LIN {X -0.090,Y -532.031,Z 1144.398,A 0.000,B 0.000,C 90.000,E1 287.692} C_DIS
LIN {X -0.142,Y -531.447,Z 1144.390,A 0.000,B 0.000,C 90.000,E1 286.260} C_DIS
LIN {X -0.170,Y -530.686,Z 1144.381,A 0.000,B 0.000,C 90.000,E1 284.537} C_DIS
LIN {X 0.098,Y -529.977,Z 1144.374,A 0.000,B 0.000,C 90.000,E1 283.355} C_DIS
LIN {X -0.145,Y -528.701,Z 1144.361,A 0.000,B 0.000,C 90.000,E1 281.074} C_DIS
LIN {X 0.034,Y -527.720,Z 1144.352,A 0.000,B 0.000,C 90.000,E1 279.321} C_DIS
LIN {X 0.037,Y -526.581,Z 1144.341,A 0.000,B 0.000,C 90.000,E1 277.296} C_DIS
LIN {X -0.057,Y -525.479,Z 1144.329,A 0.000,B 0.000,C 90.000,E1 275.277} C_DIS
LIN {X 0.247,Y -524.532,Z 1144.316,A 0.000,B 0.000,C 90.000,E1 272.922} C_DIS
LIN {X 0.030,Y -523.822,Z 1144.307,A 0.000,B 0.000,C 90.000,E1 271.203} C_DIS
LIN {X -0.209,Y -523.045,Z 1144.297,A 0.000,B 0.000,C 90.000,E1 269.484} C_DIS
LIN {X 0.023,Y -522.107,Z 1144.286,A 0.000,B 0.000,C 90.000,E1 267.421} C_DIS
LIN {X -0.216,Y -521.259,Z 1144.276,A 0.000,B 0.000,C 90.000,E1 265.698} C_DIS
LIN {X 0.175,Y -520.707,Z 1144.271,A 0.000,B 0.000,C 90.000,E1 264.780} C_DIS
LIN {X 0.024,Y -519.813,Z 1144.265,A 0.000,B 0.000,C 90.000,E1 263.628} C_DIS
LIN {X -0.168,Y -518.040,Z 1144.255,A 0.000,B 0.000,C 90.000,E1 261.894} C_DIS
LIN {X 0.162,Y -515.646,Z 1144.242,A 0.000,B 0.000,C 90.000,E1 259.511} C_DIS
LIN {X 0.113,Y -514.734,Z 1144.237,A 0.000,B 0.000,C 90.000,E1 258.634} C_DIS
LIN {X 0.008,Y -513.326,Z 1144.229,A 0.000,B 0.000,C 90.000,E1 257.173} C_DIS
LIN {X 0.011,Y -511.181,Z 1144.216,A 0.000,B 0.000,C 90.000,E1 254.810} C_DIS
LIN {X 0.078,Y -509.858,Z 1144.207,A 0.000,B 0.000,C 90.000,E1 253.323} C_DIS
LIN {X 0.266,Y -508.448,Z 1144.199,A 0.000,B 0.000,C 90.000,E1 251.819} C_DIS
LIN {X -0.151,Y -507.301,Z 1144.193,A 0.000,B 0.000,C 90.000,E1 250.678} C_DIS
LIN {X -0.143,Y -505.111,Z 1144.181,A 0.000,B 0.000,C 90.000,E1 248.592} C_DIS
LIN {X 0.211,Y -503.811,Z 1144.174,A 0.000,B 0.000,C 90.000,E1 247.358} C_DIS
LIN {X 0.078,Y -502.418,Z 1144.168,A 0.000,B 0.000,C 90.000,E1 246.177} C_DIS
LIN {X 0.129,Y -500.836,Z 1144.161,A 0.000,B 0.000,C 90.000,E1 244.973} C_DIS
LIN {X -0.230,Y -498.804,Z 1144.153,A 0.000,B 0.000,C 90.000,E1 243.512} C_DIS
LIN {X -0.124,Y -496.185,Z 1144.143,A 0.000,B 0.000,C 90.000,E1 241.691} C_DIS
LIN {X 0.057,Y -494.353,Z 1144.136,A 0.000,B 0.000,C 90.000,E1 240.461} C_DIS
LIN {X 0.033,Y -491.924,Z 1144.128,A 0.000,B 0.000,C 90.000,E1 238.948} C_DIS
LIN {X -0.041,Y -490.014,Z 1144.121,A 0.000,B 0.000,C 90.000,E1 237.740} C_DIS
LIN {X 0.192,Y -487.119,Z 1144.111,A 0.000,B 0.000,C 90.000,E1 235.881} C_DIS
LIN {X -0.043,Y -484.123,Z 1144.100,A 0.000,B 0.000,C 90.000,E1 234.069} C_DIS
LIN {X -0.266,Y -481.618,Z 1144.092,A 0.000,B 0.000,C 90.000,E1 232.557} C_DIS
LIN {X -0.058,Y -478.479,Z 1144.082,A 0.000,B 0.000,C 90.000,E1 230.678} C_DIS
LIN {X -0.148,Y -475.794,Z 1144.073,A 0.000,B 0.000,C 90.000,E1 229.138} C_DIS
LIN {X 0.171,Y -472.605,Z 1144.063,A 0.000,B 0.000,C 90.000,E1 227.229} C_DIS
LIN {X -0.067,Y -466.133,Z 1144.040,A 0.000,B 0.000,C 90.000,E1 223.176} C_DIS
LIN {X 0.091,Y -463.472,Z 1144.028,A 0.000,B 0.000,C 90.000,E1 220.943} C_DIS
LIN {X -0.133,Y -461.119,Z 1144.015,A 0.000,B 0.000,C 90.000,E1 218.749} C_DIS
LIN {X 0.111,Y -458.835,Z 1144.001,A 0.000,B 0.000,C 90.000,E1 216.171} C_DIS
LIN {X -0.031,Y -455.791,Z 1143.971,A 0.000,B 0.000,C 90.000,E1 210.747} C_DIS
LIN {X 0.088,Y -455.692,Z 1143.958,A 0.000,B 0.000,C 90.000,E1 208.487} C_DIS
LIN {X 0.068,Y -456.850,Z 1143.944,A 0.000,B 0.000,C 90.000,E1 205.924} C_DIS
LIN {X -0.111,Y -458.875,Z 1143.933,A 0.000,B 0.000,C 90.000,E1 204.027} C_DIS
LIN {X 0.171,Y -461.835,Z 1143.923,A 0.000,B 0.000,C 90.000,E1 202.078} C_DIS
LIN {X -0.117,Y -467.069,Z 1143.909,A 0.000,B 0.000,C 90.000,E1 199.577} C_DIS
LIN {X 0.019,Y -474.758,Z 1143.893,A 0.000,B 0.000,C 90.000,E1 196.732} C_DIS
LIN {X 0.039,Y -483.007,Z 1143.879,A 0.000,B 0.000,C 90.000,E1 194.245} C_DIS
LIN {X -0.161,Y -490.571,Z 1143.867,A 0.000,B 0.000,C 90.000,E1 192.119} C_DIS
LIN {X -0.200,Y -496.173,Z 1143.859,A 0.000,B 0.000,C 90.000,E1 190.602} C_DIS
LIN {X 0.210,Y -502.992,Z 1143.849,A 0.000,B 0.000,C 90.000,E1 188.746} C_DIS
LIN {X -0.174,Y -508.766,Z 1143.840,A 0.000,B 0.000,C 90.000,E1 187.296} C_DIS
LIN {X -0.020,Y -514.520,Z 1143.832,A 0.000,B 0.000,C 90.000,E1 185.796} C_DIS
LIN {X 0.198,Y -520.225,Z 1143.824,A 0.000,B 0.000,C 90.000,E1 184.302} C_DIS
LIN {X -0.001,Y -525.916,Z 1143.816,A 0.000,B 0.000,C 90.000,E1 182.865} C_DIS
LIN {X -0.163,Y -533.787,Z 1143.805,A 0.000,B 0.000,C 90.000,E1 180.859} C_DIS
LIN {X -0.160,Y -539.409,Z 1143.797,A 0.000,B 0.000,C 90.000,E1 179.427} C_DIS
LIN {X -0.042,Y -545.053,Z 1143.789,A 0.000,B 0.000,C 90.000,E1 177.993} C_DIS
LIN {X 0.235,Y -551.836,Z 1143.780,A 0.000,B 0.000,C 90.000,E1 176.274} C_DIS
LIN {X 0.255,Y -559.740,Z 1143.769,A 0.000,B 0.000,C 90.000,E1 174.318} C_DIS
LIN {X 0.285,Y -565.342,Z 1143.761,A 0.000,B 0.000,C 90.000,E1 172.932} C_DIS
LIN {X -0.147,Y -570.919,Z 1143.753,A 0.000,B 0.000,C 90.000,E1 171.602} C_DIS
LIN {X -0.038,Y -575.313,Z 1143.747,A 0.000,B 0.000,C 90.000,E1 170.500} C_DIS
LIN {X 0.132,Y -579.671,Z 1143.741,A 0.000,B 0.000,C 90.000,E1 169.398} C_DIS
LIN {X 0.137,Y -585.038,Z 1143.734,A 0.000,B 0.000,C 90.000,E1 168.049} C_DIS
LIN {X 0.240,Y -590.168,Z 1143.726,A 0.000,B 0.000,C 90.000,E1 166.700} C_DIS
LIN {X 0.150,Y -594.155,Z 1143.720,A 0.000,B 0.000,C 90.000,E1 165.644} C_DIS
LIN {X 0.260,Y -597.917,Z 1143.714,A 0.000,B 0.000,C 90.000,E1 164.574} C_DIS
LIN {X 0.033,Y -603.261,Z 1143.706,A 0.000,B 0.000,C 90.000,E1 163.015} C_DIS
LIN {X 0.184,Y -607.423,Z 1143.698,A 0.000,B 0.000,C 90.000,E1 161.692} C_DIS
LIN {X -0.115,Y -610.638,Z 1143.693,A 0.000,B 0.000,C 90.000,E1 160.678} C_DIS
LIN {X -0.224,Y -614.444,Z 1143.685,A 0.000,B 0.000,C 90.000,E1 159.390} C_DIS
LIN {X -0.269,Y -617.969,Z 1143.678,A 0.000,B 0.000,C 90.000,E1 158.103} C_DIS
LIN {X -0.027,Y -622.096,Z 1143.670,A 0.000,B 0.000,C 90.000,E1 156.538} C_DIS
LIN {X 0.317,Y -626.734,Z 1143.660,A 0.000,B 0.000,C 90.000,E1 154.717} C_DIS
LIN {X 0.137,Y -629.863,Z 1143.653,A 0.000,B 0.000,C 90.000,E1 153.461} C_DIS
LIN {X -0.282,Y -632.833,Z 1143.646,A 0.000,B 0.000,C 90.000,E1 152.231} C_DIS
LIN {X 0.209,Y -635.650,Z 1143.639,A 0.000,B 0.000,C 90.000,E1 150.923} C_DIS
LIN {X 0.198,Y -638.324,Z 1143.632,A 0.000,B 0.000,C 90.000,E1 149.665} C_DIS
LIN {X 0.227,Y -640.892,Z 1143.625,A 0.000,B 0.000,C 90.000,E1 148.408} C_DIS
LIN {X -0.310,Y -642.835,Z 1143.619,A 0.000,B 0.000,C 90.000,E1 147.454} C_DIS
LIN {X 0.003,Y -645.547,Z 1143.611,A 0.000,B 0.000,C 90.000,E1 145.928} C_DIS
LIN {X -0.053,Y -647.723,Z 1143.604,A 0.000,B 0.000,C 90.000,E1 144.689} C_DIS
LIN {X 0.262,Y -650.648,Z 1143.594,A 0.000,B 0.000,C 90.000,E1 142.924} C_DIS
LIN {X -0.006,Y -654.464,Z 1143.582,A 0.000,B 0.000,C 90.000,E1 140.723} C_DIS
LIN {X -0.168,Y -657.760,Z 1143.572,A 0.000,B 0.000,C 90.000,E1 139.013} C_DIS
LIN {X -0.321,Y -661.207,Z 1143.563,A 0.000,B 0.000,C 90.000,E1 137.310} C_DIS
LIN {X 0.053,Y -665.103,Z 1143.552,A 0.000,B 0.000,C 90.000,E1 135.324} C_DIS
LIN {X 0.059,Y -669.952,Z 1143.540,A 0.000,B 0.000,C 90.000,E1 133.137} C_DIS
LIN {X -0.245,Y -674.550,Z 1143.529,A 0.000,B 0.000,C 90.000,E1 131.229} C_DIS
LIN {X 0.115,Y -679.826,Z 1143.517,A 0.000,B 0.000,C 90.000,E1 129.036} C_DIS
LIN {X -0.068,Y -682.910,Z 1143.510,A 0.000,B 0.000,C 90.000,E1 127.855} C_DIS
LIN {X -0.046,Y -686.505,Z 1143.502,A 0.000,B 0.000,C 90.000,E1 126.423} C_DIS
LIN {X 0.011,Y -689.481,Z 1143.496,A 0.000,B 0.000,C 90.000,E1 125.231} C_DIS
LIN {X 0.332,Y -692.949,Z 1143.488,A 0.000,B 0.000,C 90.000,E1 123.785} C_DIS
LIN {X 0.112,Y -695.690,Z 1143.481,A 0.000,B 0.000,C 90.000,E1 122.625} C_DIS
LIN {X 0.029,Y -697.287,Z 1143.477,A 0.000,B 0.000,C 90.000,E1 121.926} C_DIS
LIN {X -0.158,Y -699.073,Z 1143.472,A 0.000,B 0.000,C 90.000,E1 121.003} C_DIS
LIN {X 0.233,Y -701.953,Z 1143.463,A 0.000,B 0.000,C 90.000,E1 119.333} C_DIS
LIN {X 0.053,Y -704.026,Z 1143.457,A 0.000,B 0.000,C 90.000,E1 118.180} C_DIS
LIN {X -0.337,Y -705.007,Z 1143.453,A 0.000,B 0.000,C 90.000,E1 117.513} C_DIS
LIN {X -0.099,Y -705.689,Z 1143.449,A 0.000,B 0.000,C 90.000,E1 116.796} C_DIS
LIN {X 0.120,Y -706.230,Z 1143.444,A 0.000,B 0.000,C 90.000,E1 115.848} C_DIS
LIN {X 0.058,Y -706.428,Z 1143.440,A 0.000,B 0.000,C 90.000,E1 115.155} C_DIS
LIN {X 0.001,Y -706.302,Z 1143.437,A 0.000,B 0.000,C 90.000,E1 114.695} C_DIS
LIN {X -0.001,Y -706.108,Z 1143.436,A 0.000,B 0.000,C 90.000,E1 114.463} C_DIS
LIN {X -0.064,Y -705.239,Z 1143.433,A 0.000,B 0.000,C 90.000,E1 114.003} C_DIS
LIN {X -0.062,Y -704.446,Z 1143.432,A 0.000,B 0.000,C 90.000,E1 113.770} C_DIS
LIN {X -0.418,Y -702.435,Z 1143.429,A 0.000,B 0.000,C 90.000,E1 113.334} C_DIS
LIN {X -0.279,Y -701.592,Z 1143.429,A 0.000,B 0.000,C 90.000,E1 113.206} C_DIS
LIN {X -0.004,Y -696.986,Z 1143.426,A 0.000,B 0.000,C 90.000,E1 112.717} C_DIS
LIN {X 0.133,Y -695.430,Z 1143.426,A 0.000,B 0.000,C 90.000,E1 112.589} C_DIS
LIN {X -0.198,Y -693.137,Z 1143.425,A 0.000,B 0.000,C 90.000,E1 112.514} C_DIS
LIN {X -0.032,Y -686.830,Z 1143.424,A 0.000,B 0.000,C 90.000,E1 112.280} C_DIS
LIN {X 0.249,Y -684.955,Z 1143.424,A 0.000,B 0.000,C 90.000,E1 112.206} C_DIS
LIN {X -0.087,Y -676.660,Z 1143.423,A 0.000,B 0.000,C 90.000,E1 112.153} C_DIS
LIN {X -0.125,Y -603.392,Z 1143.423,A 0.000,B 0.000,C 90.000,E1 112.153} C_DIS
LIN {X 0.313,Y -600.153,Z 1143.422,A 0.000,B 0.000,C 90.000,E1 111.897} C_DIS
LIN {X 0.268,Y -595.396,Z 1143.420,A 0.000,B 0.000,C 90.000,E1 111.535} C_DIS
LIN {X 0.101,Y -579.806,Z 1143.412,A 0.000,B 0.000,C 90.000,E1 110.174} C_DIS
LIN {X 0.002,Y -574.130,Z 1143.410,A 0.000,B 0.000,C 90.000,E1 109.704} C_DIS
LIN {X -0.219,Y -568.184,Z 1143.407,A 0.000,B 0.000,C 90.000,E1 109.268} C_DIS
LIN {X 0.008,Y -560.099,Z 1143.404,A 0.000,B 0.000,C 90.000,E1 108.725} C_DIS
LIN {X 0.116,Y -555.385,Z 1143.402,A 0.000,B 0.000,C 90.000,E1 108.417} C_DIS
LIN {X -0.140,Y -551.135,Z 1143.401,A 0.000,B 0.000,C 90.000,E1 108.109} C_DIS
LIN {X 0.243,Y -549.920,Z 1143.400,A 0.000,B 0.000,C 90.000,E1 107.873} C_DIS
LIN {X 0.200,Y -549.899,Z 1143.399,A 0.000,B 0.000,C 90.000,E1 107.873} C_DIS
LIN {X -0.090,Y -549.660,Z 1143.397,A 0.000,B 0.000,C 90.000,E1 107.457} C_DIS
LIN {X 0.223,Y -551.099,Z 1143.385,A 0.000,B 0.000,C 90.000,E1 105.190} C_DIS
LIN {X -0.033,Y -552.442,Z 1143.375,A 0.000,B 0.000,C 90.000,E1 103.536} C_DIS
LIN {X 0.272,Y -553.872,Z 1143.366,A 0.000,B 0.000,C 90.000,E1 101.827} C_DIS
LIN {X -0.161,Y -555.381,Z 1143.357,A 0.000,B 0.000,C 90.000,E1 100.197} C_DIS
LIN {X -0.146,Y -556.687,Z 1143.349,A 0.000,B 0.000,C 90.000,E1 98.803} C_DIS
LIN {X -0.052,Y -558.110,Z 1143.340,A 0.000,B 0.000,C 90.000,E1 97.125} C_DIS
LIN {X -0.071,Y -559.281,Z 1143.332,A 0.000,B 0.000,C 90.000,E1 95.739} C_DIS
LIN {X -0.040,Y -560.610,Z 1143.323,A 0.000,B 0.000,C 90.000,E1 94.073} C_DIS
LIN {X 0.118,Y -562.106,Z 1143.312,A 0.000,B 0.000,C 90.000,E1 92.121} C_DIS
LIN {X 0.179,Y -563.277,Z 1143.303,A 0.000,B 0.000,C 90.000,E1 90.458} C_DIS
LIN {X 0.038,Y -563.991,Z 1143.297,A 0.000,B 0.000,C 90.000,E1 89.370} C_DIS
LIN {X 0.137,Y -565.035,Z 1143.287,A 0.000,B 0.000,C 90.000,E1 87.707} C_DIS
LIN {X 0.253,Y -565.922,Z 1143.278,A 0.000,B 0.000,C 90.000,E1 86.045} C_DIS
LIN {X 0.204,Y -566.549,Z 1143.272,A 0.000,B 0.000,C 90.000,E1 84.951} C_DIS
LIN {X -0.126,Y -567.355,Z 1143.263,A 0.000,B 0.000,C 90.000,E1 83.337} C_DIS
LIN {X 0.195,Y -568.148,Z 1143.254,A 0.000,B 0.000,C 90.000,E1 81.659} C_DIS
LIN {X 0.167,Y -568.674,Z 1143.248,A 0.000,B 0.000,C 90.000,E1 80.566} C_DIS
LIN {X 0.139,Y -569.415,Z 1143.239,A 0.000,B 0.000,C 90.000,E1 78.926} C_DIS
LIN {X 0.017,Y -570.210,Z 1143.229,A 0.000,B 0.000,C 90.000,E1 77.297} C_DIS
LIN {X -0.215,Y -571.124,Z 1143.219,A 0.000,B 0.000,C 90.000,E1 75.408} C_DIS
LIN {X 0.093,Y -571.979,Z 1143.210,A 0.000,B 0.000,C 90.000,E1 73.740} C_DIS
LIN {X 0.237,Y -572.882,Z 1143.202,A 0.000,B 0.000,C 90.000,E1 72.362} C_DIS
LIN {X 0.203,Y -574.498,Z 1143.190,A 0.000,B 0.000,C 90.000,E1 70.188} C_DIS
LIN {X 0.074,Y -576.356,Z 1143.178,A 0.000,B 0.000,C 90.000,E1 68.028} C_DIS
LIN {X -0.004,Y -577.949,Z 1143.169,A 0.000,B 0.000,C 90.000,E1 66.410} C_DIS
LIN {X 0.177,Y -579.918,Z 1143.157,A 0.000,B 0.000,C 90.000,E1 64.229} C_DIS
LIN {X 0.128,Y -581.367,Z 1143.148,A 0.000,B 0.000,C 90.000,E1 62.615} C_DIS
LIN {X 0.110,Y -582.694,Z 1143.139,A 0.000,B 0.000,C 90.000,E1 61.001} C_DIS
LIN {X 0.022,Y -583.695,Z 1143.132,A 0.000,B 0.000,C 90.000,E1 59.665} C_DIS
LIN {X 0.093,Y -584.483,Z 1143.126,A 0.000,B 0.000,C 90.000,E1 58.584} C_DIS
LIN {X -0.097,Y -585.464,Z 1143.117,A 0.000,B 0.000,C 90.000,E1 56.993} C_DIS
LIN {X -0.127,Y -586.430,Z 1143.108,A 0.000,B 0.000,C 90.000,E1 55.388} C_DIS
LIN {X -0.132,Y -587.391,Z 1143.099,A 0.000,B 0.000,C 90.000,E1 53.783} C_DIS
LIN {X 0.150,Y -588.466,Z 1143.087,A 0.000,B 0.000,C 90.000,E1 51.618} C_DIS
LIN {X 0.227,Y -589.014,Z 1143.079,A 0.000,B 0.000,C 90.000,E1 50.275} C_DIS
LIN {X -0.078,Y -589.264,Z 1143.075,A 0.000,B 0.000,C 90.000,E1 49.504} C_DIS
LIN {X 0.015,Y -589.345,Z 1143.068,A 0.000,B 0.000,C 90.000,E1 48.162} C_DIS
LIN {X -0.286,Y -589.380,Z 1143.063,A 0.000,B 0.000,C 90.000,E1 47.391} C_DIS
LIN {X -0.243,Y -589.281,Z 1143.056,A 0.000,B 0.000,C 90.000,E1 46.053} C_DIS
LIN {X 0.034,Y -588.977,Z 1143.050,A 0.000,B 0.000,C 90.000,E1 44.960} C_DIS
LIN {X 0.305,Y -588.477,Z 1143.044,A 0.000,B 0.000,C 90.000,E1 43.866} C_DIS
LIN {X -0.253,Y -587.842,Z 1143.038,A 0.000,B 0.000,C 90.000,E1 42.852} C_DIS
LIN {X 0.011,Y -586.937,Z 1143.032,A 0.000,B 0.000,C 90.000,E1 41.757} C_DIS
LIN {X -0.130,Y -585.775,Z 1143.026,A 0.000,B 0.000,C 90.000,E1 40.701} C_DIS
LIN {X -0.286,Y -584.483,Z 1143.020,A 0.000,B 0.000,C 90.000,E1 39.644} C_DIS
LIN {X -0.010,Y -583.012,Z 1143.014,A 0.000,B 0.000,C 90.000,E1 38.543} C_DIS
LIN {X 0.244,Y -581.313,Z 1143.008,A 0.000,B 0.000,C 90.000,E1 37.443} C_DIS
LIN {X -0.051,Y -579.805,Z 1143.004,A 0.000,B 0.000,C 90.000,E1 36.664} C_DIS
LIN {X -0.019,Y -577.968,Z 1142.999,A 0.000,B 0.000,C 90.000,E1 35.851} C_DIS
LIN {X 0.121,Y -575.933,Z 1142.995,A 0.000,B 0.000,C 90.000,E1 35.025} C_DIS
LIN {X 0.244,Y -573.582,Z 1142.990,A 0.000,B 0.000,C 90.000,E1 34.199} C_DIS
LIN {X -0.268,Y -571.819,Z 1142.987,A 0.000,B 0.000,C 90.000,E1 33.706} C_DIS
LIN {X -0.188,Y -568.868,Z 1142.983,A 0.000,B 0.000,C 90.000,E1 32.880} C_DIS
LIN {X -0.255,Y -566.714,Z 1142.980,A 0.000,B 0.000,C 90.000,E1 32.339} C_DIS
LIN {X 0.247,Y -563.087,Z 1142.975,A 0.000,B 0.000,C 90.000,E1 31.465} C_DIS
LIN {X -0.051,Y -561.180,Z 1142.973,A 0.000,B 0.000,C 90.000,E1 31.082} C_DIS
LIN {X -0.100,Y -556.966,Z 1142.968,A 0.000,B 0.000,C 90.000,E1 30.256} C_DIS
LIN {X -0.108,Y -551.663,Z 1142.963,A 0.000,B 0.000,C 90.000,E1 29.283} C_DIS
LIN {X 0.180,Y -548.354,Z 1142.960,A 0.000,B 0.000,C 90.000,E1 28.693} C_DIS
LIN {X 0.192,Y -543.047,Z 1142.955,A 0.000,B 0.000,C 90.000,E1 27.847} C_DIS
LIN {X 0.276,Y -538.179,Z 1142.951,A 0.000,B 0.000,C 90.000,E1 27.129} C_DIS
LIN {X -0.264,Y -533.964,Z 1142.948,A 0.000,B 0.000,C 90.000,E1 26.616} C_DIS
LIN {X -0.085,Y -525.979,Z 1142.942,A 0.000,B 0.000,C 90.000,E1 25.591} C_DIS
LIN {X 0.136,Y -518.667,Z 1142.938,A 0.000,B 0.000,C 90.000,E1 24.719} C_DIS
LIN {X -0.240,Y -510.868,Z 1142.933,A 0.000,B 0.000,C 90.000,E1 23.898} C_DIS
LIN {X -0.290,Y -505.473,Z 1142.929,A 0.000,B 0.000,C 90.000,E1 23.334} C_DIS
LIN {X -0.178,Y -496.125,Z 1142.924,A 0.000,B 0.000,C 90.000,E1 22.386} C_DIS
LIN {X -0.186,Y -485.001,Z 1142.919,A 0.000,B 0.000,C 90.000,E1 21.354} C_DIS
LIN {X -0.172,Y -474.738,Z 1142.913,A 0.000,B 0.000,C 90.000,E1 20.429} C_DIS
LIN {X -0.046,Y -465.893,Z 1142.909,A 0.000,B 0.000,C 90.000,E1 19.631} C_DIS
LIN {X -0.103,Y -445.297,Z 1142.899,A 0.000,B 0.000,C 90.000,E1 17.764} C_DIS
LIN {X -0.196,Y -433.933,Z 1142.893,A 0.000,B 0.000,C 90.000,E1 16.677} C_DIS
LIN {X 0.162,Y -419.919,Z 1142.884,A 0.000,B 0.000,C 90.000,E1 15.134} C_DIS
LIN {X -0.059,Y -409.123,Z 1142.877,A 0.000,B 0.000,C 90.000,E1 13.883} C_DIS
LIN {X 0.012,Y -400.391,Z 1142.871,A 0.000,B 0.000,C 90.000,E1 12.703} C_DIS
LIN {X -0.168,Y -396.245,Z 1142.867,A 0.000,B 0.000,C 90.000,E1 12.063} C_DIS
LIN {X -0.136,Y -395.365,Z 1142.866,A 0.000,B 0.000,C 90.000,E1 11.883} C_DIS
LIN {X 0.033,Y -393.084,Z 1142.863,A 0.000,B 0.000,C 90.000,E1 11.299} C_DIS
LIN {X 0.166,Y -392.250,Z 1142.860,A 0.000,B 0.000,C 90.000,E1 10.838} C_DIS
LIN {X -0.164,Y -392.578,Z 1142.857,A 0.000,B 0.000,C 90.000,E1 10.310} C_DIS
LIN {X 0.148,Y -394.390,Z 1142.852,A 0.000,B 0.000,C 90.000,E1 9.378} C_DIS
LIN {X -0.047,Y -398.384,Z 1142.844,A 0.000,B 0.000,C 90.000,E1 7.992} C_DIS
LIN {X -0.142,Y -402.537,Z 1142.838,A 0.000,B 0.000,C 90.000,E1 6.777} C_DIS
LIN {X -0.179,Y -404.636,Z 1142.835,A 0.000,B 0.000,C 90.000,E1 6.258} C_DIS
LIN {X -0.181,Y -406.424,Z 1142.833,A 0.000,B 0.000,C 90.000,E1 5.910} C_DIS
LIN {X -0.202,Y -407.431,Z 1142.832,A 0.000,B 0.000,C 90.000,E1 5.739} C_DIS
LIN {X -0.185,Y -411.564,Z 1142.829,A 0.000,B 0.000,C 90.000,E1 5.220} C_DIS
LIN {X 0.112,Y -418.282,Z 1142.826,A 0.000,B 0.000,C 90.000,E1 4.645} C_DIS
LIN {X -0.120,Y -425.804,Z 1142.823,A 0.000,B 0.000,C 90.000,E1 4.131} C_DIS
LIN {X -0.206,Y -445.338,Z 1142.815,A 0.000,B 0.000,C 90.000,E1 2.751} C_DIS
LIN {X 0.142,Y -460.019,Z 1142.810,A 0.000,B 0.000,C 90.000,E1 1.718} C_DIS
LIN {X 0.110,Y -472.939,Z 1142.805,A 0.000,B 0.000,C 90.000,E1 0.859} C_DIS
LIN {X 0.037,Y -483.902,Z 1142.801,A 0.000,B 0.000,C 90.000,E1 0.115} C_DIS
LIN {X -0.218,Y -491.329,Z 1142.798,A 0.000,B 0.000,C 90.000,E1 359.599} C_DIS
LIN {X 0.157,Y -497.415,Z 1142.795,A 0.000,B 0.000,C 90.000,E1 359.083} C_DIS
LIN {X -0.096,Y -503.369,Z 1142.792,A 0.000,B 0.000,C 90.000,E1 358.625} C_DIS
LIN {X -0.060,Y -510.439,Z 1142.789,A 0.000,B 0.000,C 90.000,E1 357.993} C_DIS
LIN {X 0.234,Y -517.080,Z 1142.785,A 0.000,B 0.000,C 90.000,E1 357.306} C_DIS
LIN {X 0.111,Y -521.139,Z 1142.783,A 0.000,B 0.000,C 90.000,E1 356.906} C_DIS
LIN {X 0.124,Y -527.278,Z 1142.779,A 0.000,B 0.000,C 90.000,E1 356.216} C_DIS
LIN {X -0.126,Y -533.047,Z 1142.775,A 0.000,B 0.000,C 90.000,E1 355.527} C_DIS
LIN {X -0.073,Y -537.250,Z 1142.772,A 0.000,B 0.000,C 90.000,E1 354.951} C_DIS
LIN {X 0.245,Y -541.955,Z 1142.768,A 0.000,B 0.000,C 90.000,E1 354.204} C_DIS
LIN {X 0.063,Y -546.238,Z 1142.764,A 0.000,B 0.000,C 90.000,E1 353.514} C_DIS
LIN {X 0.240,Y -549.414,Z 1142.761,A 0.000,B 0.000,C 90.000,E1 352.932} C_DIS
LIN {X 0.120,Y -552.877,Z 1142.757,A 0.000,B 0.000,C 90.000,E1 352.243} C_DIS
LIN {X 0.105,Y -556.078,Z 1142.753,A 0.000,B 0.000,C 90.000,E1 351.546} C_DIS
LIN {X -0.018,Y -557.890,Z 1142.751,A 0.000,B 0.000,C 90.000,E1 351.141} C_DIS
LIN {X -0.243,Y -561.121,Z 1142.746,A 0.000,B 0.000,C 90.000,E1 350.330} C_DIS
LIN {X -0.180,Y -565.016,Z 1142.740,A 0.000,B 0.000,C 90.000,E1 349.218} C_DIS
LIN {X -0.169,Y -568.455,Z 1142.734,A 0.000,B 0.000,C 90.000,E1 348.117} C_DIS
LIN {X 0.315,Y -572.366,Z 1142.726,A 0.000,B 0.000,C 90.000,E1 346.700} C_DIS
LIN {X -0.019,Y -575.337,Z 1142.720,A 0.000,B 0.000,C 90.000,E1 345.644} C_DIS
LIN {X 0.177,Y -577.458,Z 1142.716,A 0.000,B 0.000,C 90.000,E1 344.810} C_DIS
LIN {X 0.089,Y -581.463,Z 1142.707,A 0.000,B 0.000,C 90.000,E1 343.196} C_DIS
LIN {X -0.140,Y -584.612,Z 1142.699,A 0.000,B 0.000,C 90.000,E1 341.873} C_DIS
LIN {X -0.323,Y -587.465,Z 1142.692,A 0.000,B 0.000,C 90.000,E1 340.550} C_DIS
LIN {X 0.062,Y -589.511,Z 1142.686,A 0.000,B 0.000,C 90.000,E1 339.444} C_DIS
LIN {X 0.045,Y -590.917,Z 1142.681,A 0.000,B 0.000,C 90.000,E1 338.646} C_DIS
LIN {X 0.042,Y -592.188,Z 1142.677,A 0.000,B 0.000,C 90.000,E1 337.847} C_DIS
LIN {X -0.153,Y -593.698,Z 1142.670,A 0.000,B 0.000,C 90.000,E1 336.538} C_DIS
LIN {X -0.139,Y -594.363,Z 1142.665,A 0.000,B 0.000,C 90.000,E1 335.741} C_DIS
LIN {X 0.121,Y -594.853,Z 1142.661,A 0.000,B 0.000,C 90.000,E1 334.921} C_DIS
LIN {X -0.061,Y -595.044,Z 1142.658,A 0.000,B 0.000,C 90.000,E1 334.409} C_DIS
LIN {X 0.204,Y -594.961,Z 1142.653,A 0.000,B 0.000,C 90.000,E1 333.589} C_DIS
LIN {X 0.024,Y -594.736,Z 1142.651,A 0.000,B 0.000,C 90.000,E1 333.076} C_DIS
LIN {X 0.025,Y -594.126,Z 1142.646,A 0.000,B 0.000,C 90.000,E1 332.281} C_DIS
LIN {X -0.253,Y -593.182,Z 1142.642,A 0.000,B 0.000,C 90.000,E1 331.513} C_DIS
LIN {X -0.159,Y -592.444,Z 1142.639,A 0.000,B 0.000,C 90.000,E1 330.973} C_DIS
LIN {X 0.158,Y -591.429,Z 1142.636,A 0.000,B 0.000,C 90.000,E1 330.411} C_DIS
LIN {X 0.242,Y -590.245,Z 1142.633,A 0.000,B 0.000,C 90.000,E1 329.871} C_DIS
LIN {X 0.206,Y -588.156,Z 1142.628,A 0.000,B 0.000,C 90.000,E1 329.076} C_DIS
LIN {X 0.146,Y -585.412,Z 1142.624,A 0.000,B 0.000,C 90.000,E1 328.280} C_DIS
LIN {X -0.125,Y -582.067,Z 1142.619,A 0.000,B 0.000,C 90.000,E1 327.502} C_DIS
LIN {X -0.175,Y -578.679,Z 1142.616,A 0.000,B 0.000,C 90.000,E1 326.834} C_DIS
LIN {X 0.058,Y -574.838,Z 1142.612,A 0.000,B 0.000,C 90.000,E1 326.135} C_DIS
LIN {X 0.028,Y -571.479,Z 1142.609,A 0.000,B 0.000,C 90.000,E1 325.595} C_DIS
LIN {X 0.092,Y -565.742,Z 1142.604,A 0.000,B 0.000,C 90.000,E1 324.769} C_DIS
LIN {X 0.098,Y -562.631,Z 1142.602,A 0.000,B 0.000,C 90.000,E1 324.356} C_DIS
LIN {X 0.012,Y -558.280,Z 1142.599,A 0.000,B 0.000,C 90.000,E1 323.829} C_DIS
LIN {X -0.059,Y -550.998,Z 1142.594,A 0.000,B 0.000,C 90.000,E1 323.004} C_DIS
LIN {X -0.221,Y -543.411,Z 1142.590,A 0.000,B 0.000,C 90.000,E1 322.190} C_DIS
LIN {X 0.062,Y -533.181,Z 1142.584,A 0.000,B 0.000,C 90.000,E1 321.045} C_DIS
LIN {X -0.156,Y -529.759,Z 1142.581,A 0.000,B 0.000,C 90.000,E1 320.642} C_DIS
LIN {X -0.014,Y -527.084,Z 1142.579,A 0.000,B 0.000,C 90.000,E1 320.194} C_DIS
LIN {X 0.245,Y -524.363,Z 1142.575,A 0.000,B 0.000,C 90.000,E1 319.542} C_DIS
LIN {X 0.258,Y -522.935,Z 1142.572,A 0.000,B 0.000,C 90.000,E1 318.933} C_DIS
LIN {X -0.035,Y -522.501,Z 1142.570,A 0.000,B 0.000,C 90.000,E1 318.528} C_DIS
LIN {X -0.085,Y -522.092,Z 1142.568,A 0.000,B 0.000,C 90.000,E1 318.243} C_DIS
LIN {X 0.073,Y -521.821,Z 1142.562,A 0.000,B 0.000,C 90.000,E1 317.067} C_DIS
LIN {X -0.051,Y -522.532,Z 1142.550,A 0.000,B 0.000,C 90.000,E1 315.040} C_DIS
LIN {X -0.100,Y -523.121,Z 1142.541,A 0.000,B 0.000,C 90.000,E1 313.299} C_DIS
LIN {X -0.239,Y -523.992,Z 1142.528,A 0.000,B 0.000,C 90.000,E1 310.987} C_DIS
LIN {X 0.185,Y -524.838,Z 1142.518,A 0.000,B 0.000,C 90.000,E1 309.197} C_DIS
LIN {X 0.332,Y -525.708,Z 1142.510,A 0.000,B 0.000,C 90.000,E1 307.729} C_DIS
LIN {X 0.085,Y -527.153,Z 1142.497,A 0.000,B 0.000,C 90.000,E1 305.438} C_DIS
LIN {X 0.048,Y -528.318,Z 1142.487,A 0.000,B 0.000,C 90.000,E1 303.706} C_DIS
LIN {X 0.138,Y -529.857,Z 1142.474,A 0.000,B 0.000,C 90.000,E1 301.386} C_DIS
LIN {X 0.080,Y -530.913,Z 1142.467,A 0.000,B 0.000,C 90.000,E1 299.951} C_DIS
LIN {X 0.018,Y -532.044,Z 1142.457,A 0.000,B 0.000,C 90.000,E1 298.231} C_DIS
LIN {X 0.187,Y -532.731,Z 1142.447,A 0.000,B 0.000,C 90.000,E1 296.488} C_DIS
LIN {X -0.065,Y -532.988,Z 1142.439,A 0.000,B 0.000,C 90.000,E1 295.079} C_DIS
LIN {X 0.143,Y -533.018,Z 1142.430,A 0.000,B 0.000,C 90.000,E1 293.334} C_DIS
LIN {X -0.137,Y -533.008,Z 1142.419,A 0.000,B 0.000,C 90.000,E1 291.354} C_DIS
LIN {X 0.176,Y -532.892,Z 1142.411,A 0.000,B 0.000,C 90.000,E1 289.885} C_DIS
LIN {X -0.197,Y -532.526,Z 1142.403,A 0.000,B 0.000,C 90.000,E1 288.489} C_DIS
LIN {X 0.215,Y -532.294,Z 1142.398,A 0.000,B 0.000,C 90.000,E1 287.583} C_DIS
LIN {X 0.176,Y -531.727,Z 1142.390,A 0.000,B 0.000,C 90.000,E1 286.150} C_DIS
LIN {X 0.125,Y -531.112,Z 1142.382,A 0.000,B 0.000,C 90.000,E1 284.717} C_DIS
LIN {X -0.114,Y -530.434,Z 1142.375,A 0.000,B 0.000,C 90.000,E1 283.592} C_DIS
LIN {X 0.282,Y -529.188,Z 1142.363,A 0.000,B 0.000,C 90.000,E1 281.243} C_DIS
LIN {X -0.117,Y -528.034,Z 1142.351,A 0.000,B 0.000,C 90.000,E1 279.265} C_DIS
LIN {X -0.104,Y -526.904,Z 1142.340,A 0.000,B 0.000,C 90.000,E1 277.239} C_DIS
LIN {X -0.187,Y -525.837,Z 1142.329,A 0.000,B 0.000,C 90.000,E1 275.220} C_DIS
LIN {X 0.140,Y -525.017,Z 1142.318,A 0.000,B 0.000,C 90.000,E1 273.154} C_DIS
LIN {X -0.041,Y -524.286,Z 1142.308,A 0.000,B 0.000,C 90.000,E1 271.432} C_DIS
LIN {X 0.213,Y -523.392,Z 1142.297,A 0.000,B 0.000,C 90.000,E1 269.370} C_DIS
LIN {X -0.026,Y -522.588,Z 1142.287,A 0.000,B 0.000,C 90.000,E1 267.650} C_DIS
LIN {X 0.271,Y -521.737,Z 1142.277,A 0.000,B 0.000,C 90.000,E1 265.869} C_DIS
LIN {X 0.092,Y -521.010,Z 1142.271,A 0.000,B 0.000,C 90.000,E1 264.723} C_DIS
LIN {X -0.056,Y -520.131,Z 1142.264,A 0.000,B 0.000,C 90.000,E1 263.571} C_DIS
LIN {X -0.242,Y -518.359,Z 1142.255,A 0.000,B 0.000,C 90.000,E1 261.837} C_DIS
LIN {X 0.093,Y -515.979,Z 1142.242,A 0.000,B 0.000,C 90.000,E1 259.454} C_DIS
LIN {X -0.032,Y -513.939,Z 1142.230,A 0.000,B 0.000,C 90.000,E1 257.409} C_DIS
LIN {X -0.047,Y -511.513,Z 1142.215,A 0.000,B 0.000,C 90.000,E1 254.755} C_DIS
LIN {X 0.122,Y -509.903,Z 1142.205,A 0.000,B 0.000,C 90.000,E1 252.960} C_DIS
LIN {X -0.234,Y -508.164,Z 1142.196,A 0.000,B 0.000,C 90.000,E1 251.221} C_DIS
LIN {X 0.084,Y -506.605,Z 1142.187,A 0.000,B 0.000,C 90.000,E1 249.699} C_DIS
LIN {X -0.105,Y -505.062,Z 1142.179,A 0.000,B 0.000,C 90.000,E1 248.230} C_DIS
LIN {X -0.137,Y -503.391,Z 1142.171,A 0.000,B 0.000,C 90.000,E1 246.741} C_DIS
LIN {X -0.072,Y -501.874,Z 1142.164,A 0.000,B 0.000,C 90.000,E1 245.537} C_DIS
LIN {X 0.102,Y -499.417,Z 1142.154,A 0.000,B 0.000,C 90.000,E1 243.717} C_DIS
LIN {X -0.065,Y -497.244,Z 1142.146,A 0.000,B 0.000,C 90.000,E1 242.231} C_DIS
LIN {X -0.031,Y -495.016,Z 1142.137,A 0.000,B 0.000,C 90.000,E1 240.717} C_DIS
LIN {X -0.038,Y -492.557,Z 1142.129,A 0.000,B 0.000,C 90.000,E1 239.203} C_DIS
LIN {X -0.098,Y -490.632,Z 1142.122,A 0.000,B 0.000,C 90.000,E1 237.995} C_DIS
LIN {X -0.115,Y -487.740,Z 1142.112,A 0.000,B 0.000,C 90.000,E1 236.167} C_DIS
LIN {X 0.117,Y -485.216,Z 1142.104,A 0.000,B 0.000,C 90.000,E1 234.609} C_DIS
LIN {X 0.127,Y -482.196,Z 1142.093,A 0.000,B 0.000,C 90.000,E1 232.763} C_DIS
LIN {X -0.021,Y -479.025,Z 1142.083,A 0.000,B 0.000,C 90.000,E1 230.928} C_DIS
LIN {X -0.038,Y -476.347,Z 1142.074,A 0.000,B 0.000,C 90.000,E1 229.380} C_DIS
LIN {X 0.289,Y -473.122,Z 1142.064,A 0.000,B 0.000,C 90.000,E1 227.472} C_DIS
LIN {X 0.072,Y -466.551,Z 1142.041,A 0.000,B 0.000,C 90.000,E1 223.419} C_DIS
LIN {X -0.054,Y -463.402,Z 1142.027,A 0.000,B 0.000,C 90.000,E1 220.906} C_DIS
LIN {X 0.066,Y -460.969,Z 1142.015,A 0.000,B 0.000,C 90.000,E1 218.669} C_DIS
LIN {X -0.071,Y -458.567,Z 1142.001,A 0.000,B 0.000,C 90.000,E1 216.137} C_DIS
LIN {X -0.189,Y -455.070,Z 1141.965,A 0.000,B 0.000,C 90.000,E1 209.745} C_DIS
LIN {X 0.088,Y -455.271,Z 1141.953,A 0.000,B 0.000,C 90.000,E1 207.462} C_DIS
LIN {X 0.066,Y -456.319,Z 1141.942,A 0.000,B 0.000,C 90.000,E1 205.540} C_DIS
LIN {X 0.058,Y -457.635,Z 1141.935,A 0.000,B 0.000,C 90.000,E1 204.259} C_DIS
LIN {X 0.125,Y -460.431,Z 1141.924,A 0.000,B 0.000,C 90.000,E1 202.333} C_DIS
LIN {X -0.108,Y -466.322,Z 1141.908,A 0.000,B 0.000,C 90.000,E1 199.504} C_DIS
LIN {X -0.148,Y -474.131,Z 1141.893,A 0.000,B 0.000,C 90.000,E1 196.677} C_DIS
LIN {X 0.004,Y -481.384,Z 1141.880,A 0.000,B 0.000,C 90.000,E1 194.481} C_DIS
LIN {X -0.115,Y -487.895,Z 1141.870,A 0.000,B 0.000,C 90.000,E1 192.647} C_DIS
LIN {X 0.182,Y -494.623,Z 1141.860,A 0.000,B 0.000,C 90.000,E1 190.782} C_DIS
LIN {X 0.150,Y -501.517,Z 1141.850,A 0.000,B 0.000,C 90.000,E1 188.973} C_DIS
LIN {X 0.111,Y -508.494,Z 1141.840,A 0.000,B 0.000,C 90.000,E1 187.182} C_DIS
LIN {X -0.242,Y -514.258,Z 1141.832,A 0.000,B 0.000,C 90.000,E1 185.739} C_DIS
LIN {X 0.037,Y -518.854,Z 1141.825,A 0.000,B 0.000,C 90.000,E1 184.531} C_DIS
LIN {X -0.236,Y -525.746,Z 1141.816,A 0.000,B 0.000,C 90.000,E1 182.808} C_DIS
LIN {X 0.130,Y -533.671,Z 1141.804,A 0.000,B 0.000,C 90.000,E1 180.745} C_DIS
LIN {X 0.146,Y -540.483,Z 1141.795,A 0.000,B 0.000,C 90.000,E1 179.026} C_DIS
LIN {X -0.259,Y -546.191,Z 1141.787,A 0.000,B 0.000,C 90.000,E1 177.650} C_DIS
LIN {X -0.019,Y -551.878,Z 1141.779,A 0.000,B 0.000,C 90.000,E1 176.216} C_DIS
LIN {X -0.073,Y -558.697,Z 1141.770,A 0.000,B 0.000,C 90.000,E1 174.546} C_DIS
LIN {X -0.127,Y -564.374,Z 1141.762,A 0.000,B 0.000,C 90.000,E1 173.166} C_DIS
LIN {X 0.157,Y -571.124,Z 1141.753,A 0.000,B 0.000,C 90.000,E1 171.489} C_DIS
LIN {X 0.113,Y -577.816,Z 1141.744,A 0.000,B 0.000,C 90.000,E1 169.859} C_DIS
LIN {X 0.209,Y -584.252,Z 1141.735,A 0.000,B 0.000,C 90.000,E1 168.229} C_DIS
LIN {X -0.279,Y -589.481,Z 1141.727,A 0.000,B 0.000,C 90.000,E1 166.937} C_DIS
LIN {X 0.036,Y -594.476,Z 1141.720,A 0.000,B 0.000,C 90.000,E1 165.574} C_DIS
LIN {X -0.002,Y -598.223,Z 1141.714,A 0.000,B 0.000,C 90.000,E1 164.519} C_DIS
LIN {X 0.051,Y -602.692,Z 1141.707,A 0.000,B 0.000,C 90.000,E1 163.196} C_DIS
LIN {X 0.191,Y -606.936,Z 1141.699,A 0.000,B 0.000,C 90.000,E1 161.873} C_DIS
LIN {X -0.176,Y -610.922,Z 1141.692,A 0.000,B 0.000,C 90.000,E1 160.604} C_DIS
LIN {X -0.230,Y -613.999,Z 1141.686,A 0.000,B 0.000,C 90.000,E1 159.571} C_DIS
LIN {X -0.279,Y -617.540,Z 1141.679,A 0.000,B 0.000,C 90.000,E1 158.284} C_DIS
LIN {X -0.298,Y -622.361,Z 1141.669,A 0.000,B 0.000,C 90.000,E1 156.485} C_DIS
LIN {X 0.042,Y -626.973,Z 1141.659,A 0.000,B 0.000,C 90.000,E1 154.665} C_DIS
LIN {X 0.140,Y -630.064,Z 1141.652,A 0.000,B 0.000,C 90.000,E1 153.384} C_DIS
LIN {X -0.269,Y -632.999,Z 1141.645,A 0.000,B 0.000,C 90.000,E1 152.153} C_DIS
LIN {X 0.231,Y -635.788,Z 1141.638,A 0.000,B 0.000,C 90.000,E1 150.845} C_DIS
LIN {X -0.097,Y -638.449,Z 1141.631,A 0.000,B 0.000,C 90.000,E1 149.616} C_DIS
LIN {X 0.263,Y -641.018,Z 1141.624,A 0.000,B 0.000,C 90.000,E1 148.329} C_DIS
LIN {X -0.270,Y -642.921,Z 1141.619,A 0.000,B 0.000,C 90.000,E1 147.375} C_DIS
LIN {X 0.169,Y -645.182,Z 1141.612,A 0.000,B 0.000,C 90.000,E1 146.087} C_DIS
LIN {X 0.049,Y -646.958,Z 1141.606,A 0.000,B 0.000,C 90.000,E1 145.102} C_DIS
LIN {X -0.084,Y -649.470,Z 1141.598,A 0.000,B 0.000,C 90.000,E1 143.623} C_DIS
LIN {X -0.225,Y -651.562,Z 1141.591,A 0.000,B 0.000,C 90.000,E1 142.396} C_DIS
LIN {X 0.061,Y -654.569,Z 1141.581,A 0.000,B 0.000,C 90.000,E1 140.642} C_DIS
LIN {X -0.096,Y -657.858,Z 1141.572,A 0.000,B 0.000,C 90.000,E1 138.933} C_DIS
LIN {X -0.245,Y -661.293,Z 1141.562,A 0.000,B 0.000,C 90.000,E1 137.229} C_DIS
LIN {X 0.138,Y -664.719,Z 1141.553,A 0.000,B 0.000,C 90.000,E1 135.486} C_DIS
LIN {X 0.135,Y -669.504,Z 1141.541,A 0.000,B 0.000,C 90.000,E1 133.299} C_DIS
LIN {X -0.178,Y -674.082,Z 1141.530,A 0.000,B 0.000,C 90.000,E1 131.391} C_DIS
LIN {X 0.013,Y -677.561,Z 1141.522,A 0.000,B 0.000,C 90.000,E1 129.930} C_DIS
LIN {X -0.010,Y -682.458,Z 1141.511,A 0.000,B 0.000,C 90.000,E1 128.016} C_DIS
LIN {X 0.010,Y -686.082,Z 1141.503,A 0.000,B 0.000,C 90.000,E1 126.583} C_DIS
LIN {X 0.096,Y -689.618,Z 1141.495,A 0.000,B 0.000,C 90.000,E1 125.152} C_DIS
LIN {X 0.417,Y -693.072,Z 1141.488,A 0.000,B 0.000,C 90.000,E1 123.706} C_DIS
LIN {X 0.195,Y -695.829,Z 1141.481,A 0.000,B 0.000,C 90.000,E1 122.546} C_DIS
LIN {X 0.357,Y -697.856,Z 1141.476,A 0.000,B 0.000,C 90.000,E1 121.592} C_DIS
LIN {X 0.180,Y -699.599,Z 1141.470,A 0.000,B 0.000,C 90.000,E1 120.669} C_DIS
LIN {X -0.100,Y -702.912,Z 1141.460,A 0.000,B 0.000,C 90.000,E1 118.821} C_DIS
LIN {X 0.124,Y -704.123,Z 1141.456,A 0.000,B 0.000,C 90.000,E1 118.103} C_DIS
LIN {X 0.017,Y -705.266,Z 1141.451,A 0.000,B 0.000,C 90.000,E1 117.180} C_DIS
LIN {X -0.352,Y -705.677,Z 1141.448,A 0.000,B 0.000,C 90.000,E1 116.744} C_DIS
LIN {X -0.129,Y -706.229,Z 1141.443,A 0.000,B 0.000,C 90.000,E1 115.796} C_DIS
LIN {X 0.112,Y -706.382,Z 1141.439,A 0.000,B 0.000,C 90.000,E1 115.079} C_DIS
LIN {X -0.242,Y -706.258,Z 1141.437,A 0.000,B 0.000,C 90.000,E1 114.643} C_DIS
LIN {X 0.051,Y -705.507,Z 1141.434,A 0.000,B 0.000,C 90.000,E1 114.155} C_DIS
LIN {X -0.303,Y -705.045,Z 1141.433,A 0.000,B 0.000,C 90.000,E1 113.951} C_DIS
LIN {X -0.014,Y -703.162,Z 1141.430,A 0.000,B 0.000,C 90.000,E1 113.462} C_DIS
LIN {X 0.266,Y -701.949,Z 1141.429,A 0.000,B 0.000,C 90.000,E1 113.206} C_DIS
LIN {X -0.088,Y -697.456,Z 1141.427,A 0.000,B 0.000,C 90.000,E1 112.770} C_DIS
LIN {X 0.046,Y -696.133,Z 1141.426,A 0.000,B 0.000,C 90.000,E1 112.642} C_DIS
LIN {X 0.178,Y -694.007,Z 1141.425,A 0.000,B 0.000,C 90.000,E1 112.514} C_DIS
LIN {X -0.201,Y -685.685,Z 1141.424,A 0.000,B 0.000,C 90.000,E1 112.259} C_DIS
LIN {X -0.030,Y -683.042,Z 1141.423,A 0.000,B 0.000,C 90.000,E1 112.206} C_DIS
LIN {X -0.094,Y -676.898,Z 1141.423,A 0.000,B 0.000,C 90.000,E1 112.153} C_DIS
LIN {X -0.130,Y -603.382,Z 1141.423,A 0.000,B 0.000,C 90.000,E1 112.153} C_DIS
LIN {X -0.168,Y -600.249,Z 1141.422,A 0.000,B 0.000,C 90.000,E1 111.950} C_DIS
LIN {X -0.201,Y -595.464,Z 1141.420,A 0.000,B 0.000,C 90.000,E1 111.589} C_DIS
LIN {X 0.102,Y -580.049,Z 1141.412,A 0.000,B 0.000,C 90.000,E1 110.194} C_DIS
LIN {X 0.180,Y -574.381,Z 1141.410,A 0.000,B 0.000,C 90.000,E1 109.704} C_DIS
LIN {X -0.082,Y -568.432,Z 1141.407,A 0.000,B 0.000,C 90.000,E1 109.268} C_DIS
LIN {X 0.105,Y -560.248,Z 1141.404,A 0.000,B 0.000,C 90.000,E1 108.725} C_DIS
LIN {X 0.224,Y -555.521,Z 1141.402,A 0.000,B 0.000,C 90.000,E1 108.417} C_DIS
LIN {X -0.098,Y -551.143,Z 1141.401,A 0.000,B 0.000,C 90.000,E1 108.109} C_DIS
LIN {X 0.200,Y -549.855,Z 1141.399,A 0.000,B 0.000,C 90.000,E1 107.873} C_DIS
LIN {X 0.158,Y -549.834,Z 1141.399,A 0.000,B 0.000,C 90.000,E1 107.873} C_DIS
LIN {X -0.049,Y -549.599,Z 1141.397,A 0.000,B 0.000,C 90.000,E1 107.457} C_DIS
LIN {X 0.263,Y -551.037,Z 1141.385,A 0.000,B 0.000,C 90.000,E1 105.190} C_DIS
LIN {X -0.111,Y -552.135,Z 1141.377,A 0.000,B 0.000,C 90.000,E1 103.828} C_DIS
LIN {X 0.186,Y -553.591,Z 1141.367,A 0.000,B 0.000,C 90.000,E1 102.119} C_DIS
LIN {X -0.127,Y -555.287,Z 1141.357,A 0.000,B 0.000,C 90.000,E1 100.197} C_DIS
LIN {X -0.112,Y -556.594,Z 1141.349,A 0.000,B 0.000,C 90.000,E1 98.803} C_DIS
LIN {X -0.022,Y -558.016,Z 1141.340,A 0.000,B 0.000,C 90.000,E1 97.125} C_DIS
LIN {X 0.035,Y -559.422,Z 1141.330,A 0.000,B 0.000,C 90.000,E1 95.454} C_DIS
LIN {X 0.114,Y -560.774,Z 1141.321,A 0.000,B 0.000,C 90.000,E1 93.784} C_DIS
LIN {X 0.146,Y -562.052,Z 1141.312,A 0.000,B 0.000,C 90.000,E1 92.121} C_DIS
LIN {X -0.254,Y -563.411,Z 1141.301,A 0.000,B 0.000,C 90.000,E1 90.229} C_DIS
LIN {X 0.170,Y -564.054,Z 1141.295,A 0.000,B 0.000,C 90.000,E1 89.083} C_DIS
LIN {X 0.161,Y -564.958,Z 1141.287,A 0.000,B 0.000,C 90.000,E1 87.707} C_DIS
LIN {X -0.142,Y -565.983,Z 1141.277,A 0.000,B 0.000,C 90.000,E1 85.812} C_DIS
LIN {X 0.225,Y -566.452,Z 1141.272,A 0.000,B 0.000,C 90.000,E1 84.951} C_DIS
LIN {X -0.108,Y -567.258,Z 1141.263,A 0.000,B 0.000,C 90.000,E1 83.337} C_DIS
LIN {X -0.258,Y -568.156,Z 1141.252,A 0.000,B 0.000,C 90.000,E1 81.432} C_DIS
LIN {X -0.200,Y -568.662,Z 1141.246,A 0.000,B 0.000,C 90.000,E1 80.330} C_DIS
LIN {X -0.335,Y -569.367,Z 1141.237,A 0.000,B 0.000,C 90.000,E1 78.701} C_DIS
LIN {X 0.027,Y -570.082,Z 1141.229,A 0.000,B 0.000,C 90.000,E1 77.297} C_DIS
LIN {X -0.026,Y -570.669,Z 1141.222,A 0.000,B 0.000,C 90.000,E1 75.936} C_DIS
LIN {X -0.245,Y -571.219,Z 1141.216,A 0.000,B 0.000,C 90.000,E1 74.866} C_DIS
LIN {X 0.096,Y -571.853,Z 1141.210,A 0.000,B 0.000,C 90.000,E1 73.740} C_DIS
LIN {X -0.130,Y -572.922,Z 1141.201,A 0.000,B 0.000,C 90.000,E1 72.127} C_DIS
LIN {X 0.025,Y -574.588,Z 1141.189,A 0.000,B 0.000,C 90.000,E1 69.934} C_DIS
LIN {X -0.308,Y -576.510,Z 1141.177,A 0.000,B 0.000,C 90.000,E1 67.794} C_DIS
LIN {X -0.013,Y -577.835,Z 1141.169,A 0.000,B 0.000,C 90.000,E1 66.410} C_DIS
LIN {X -0.215,Y -579.554,Z 1141.158,A 0.000,B 0.000,C 90.000,E1 64.537} C_DIS
LIN {X 0.114,Y -581.244,Z 1141.148,A 0.000,B 0.000,C 90.000,E1 62.615} C_DIS
LIN {X 0.094,Y -582.554,Z 1141.139,A 0.000,B 0.000,C 90.000,E1 61.001} C_DIS
LIN {X 0.003,Y -583.515,Z 1141.131,A 0.000,B 0.000,C 90.000,E1 59.665} C_DIS
LIN {X 0.071,Y -584.335,Z 1141.126,A 0.000,B 0.000,C 90.000,E1 58.584} C_DIS
LIN {X 0.197,Y -585.289,Z 1141.117,A 0.000,B 0.000,C 90.000,E1 56.962} C_DIS
LIN {X 0.034,Y -586.407,Z 1141.106,A 0.000,B 0.000,C 90.000,E1 55.102} C_DIS
LIN {X -0.166,Y -587.201,Z 1141.099,A 0.000,B 0.000,C 90.000,E1 53.783} C_DIS
LIN {X 0.111,Y -588.258,Z 1141.087,A 0.000,B 0.000,C 90.000,E1 51.618} C_DIS
LIN {X -0.069,Y -588.916,Z 1141.078,A 0.000,B 0.000,C 90.000,E1 50.033} C_DIS
LIN {X 0.269,Y -589.067,Z 1141.072,A 0.000,B 0.000,C 90.000,E1 48.933} C_DIS
LIN {X -0.092,Y -589.107,Z 1141.065,A 0.000,B 0.000,C 90.000,E1 47.634} C_DIS
LIN {X -0.057,Y -589.007,Z 1141.057,A 0.000,B 0.000,C 90.000,E1 46.296} C_DIS
LIN {X -0.199,Y -588.771,Z 1141.051,A 0.000,B 0.000,C 90.000,E1 45.243} C_DIS
LIN {X -0.345,Y -588.318,Z 1141.045,A 0.000,B 0.000,C 90.000,E1 44.190} C_DIS
LIN {X -0.322,Y -587.521,Z 1141.038,A 0.000,B 0.000,C 90.000,E1 42.852} C_DIS
LIN {X 0.190,Y -586.883,Z 1141.033,A 0.000,B 0.000,C 90.000,E1 42.000} C_DIS
LIN {X 0.050,Y -585.730,Z 1141.028,A 0.000,B 0.000,C 90.000,E1 40.943} C_DIS
LIN {X -0.369,Y -584.091,Z 1141.020,A 0.000,B 0.000,C 90.000,E1 39.644} C_DIS
LIN {X -0.099,Y -582.612,Z 1141.014,A 0.000,B 0.000,C 90.000,E1 38.543} C_DIS
LIN {X 0.149,Y -580.872,Z 1141.008,A 0.000,B 0.000,C 90.000,E1 37.443} C_DIS
LIN {X -0.150,Y -579.319,Z 1141.004,A 0.000,B 0.000,C 90.000,E1 36.664} C_DIS
LIN {X 0.184,Y -578.168,Z 1141.001,A 0.000,B 0.000,C 90.000,E1 36.091} C_DIS
LIN {X 0.013,Y -575.417,Z 1140.995,A 0.000,B 0.000,C 90.000,E1 35.025} C_DIS
LIN {X 0.131,Y -573.039,Z 1140.990,A 0.000,B 0.000,C 90.000,E1 34.199} C_DIS
LIN {X 0.092,Y -571.264,Z 1140.987,A 0.000,B 0.000,C 90.000,E1 33.658} C_DIS
LIN {X 0.288,Y -567.182,Z 1140.981,A 0.000,B 0.000,C 90.000,E1 32.546} C_DIS
LIN {X 0.016,Y -563.709,Z 1140.976,A 0.000,B 0.000,C 90.000,E1 31.750} C_DIS
LIN {X 0.102,Y -560.487,Z 1140.973,A 0.000,B 0.000,C 90.000,E1 31.052} C_DIS
LIN {X 0.239,Y -556.254,Z 1140.968,A 0.000,B 0.000,C 90.000,E1 30.207} C_DIS
LIN {X -0.258,Y -550.870,Z 1140.963,A 0.000,B 0.000,C 90.000,E1 29.283} C_DIS
LIN {X 0.143,Y -548.424,Z 1140.960,A 0.000,B 0.000,C 90.000,E1 28.821} C_DIS
LIN {X 0.029,Y -542.219,Z 1140.955,A 0.000,B 0.000,C 90.000,E1 27.847} C_DIS
LIN {X 0.108,Y -537.288,Z 1140.951,A 0.000,B 0.000,C 90.000,E1 27.129} C_DIS
LIN {X 0.040,Y -533.048,Z 1140.948,A 0.000,B 0.000,C 90.000,E1 26.565} C_DIS
LIN {X 0.206,Y -525.025,Z 1140.942,A 0.000,B 0.000,C 90.000,E1 25.540} C_DIS
LIN {X -0.038,Y -517.456,Z 1140.937,A 0.000,B 0.000,C 90.000,E1 24.695} C_DIS
LIN {X 0.278,Y -511.094,Z 1140.933,A 0.000,B 0.000,C 90.000,E1 23.951} C_DIS
LIN {X 0.282,Y -505.785,Z 1140.930,A 0.000,B 0.000,C 90.000,E1 23.387} C_DIS
LIN {X 0.135,Y -496.381,Z 1140.925,A 0.000,B 0.000,C 90.000,E1 22.461} C_DIS
LIN {X 0.012,Y -486.230,Z 1140.920,A 0.000,B 0.000,C 90.000,E1 21.535} C_DIS
LIN {X -0.046,Y -477.415,Z 1140.915,A 0.000,B 0.000,C 90.000,E1 20.737} C_DIS
LIN {X -0.090,Y -465.449,Z 1140.909,A 0.000,B 0.000,C 90.000,E1 19.685} C_DIS
LIN {X 0.029,Y -448.381,Z 1140.901,A 0.000,B 0.000,C 90.000,E1 18.127} C_DIS
LIN {X -0.195,Y -432.527,Z 1140.892,A 0.000,B 0.000,C 90.000,E1 16.622} C_DIS
LIN {X 0.033,Y -419.950,Z 1140.885,A 0.000,B 0.000,C 90.000,E1 15.245} C_DIS
LIN {X 0.121,Y -409.109,Z 1140.878,A 0.000,B 0.000,C 90.000,E1 13.953} C_DIS
LIN {X 0.126,Y -401.515,Z 1140.872,A 0.000,B 0.000,C 90.000,E1 12.939} C_DIS
LIN {X 0.156,Y -398.052,Z 1140.869,A 0.000,B 0.000,C 90.000,E1 12.411} C_DIS
LIN {X 0.110,Y -395.326,Z 1140.867,A 0.000,B 0.000,C 90.000,E1 11.951} C_DIS
LIN {X -0.144,Y -393.085,Z 1140.863,A 0.000,B 0.000,C 90.000,E1 11.422} C_DIS
LIN {X 0.015,Y -392.208,Z 1140.861,A 0.000,B 0.000,C 90.000,E1 10.950} C_DIS
LIN {X 0.147,Y -392.540,Z 1140.857,A 0.000,B 0.000,C 90.000,E1 10.310} C_DIS
LIN {X 0.197,Y -393.631,Z 1140.854,A 0.000,B 0.000,C 90.000,E1 9.726} C_DIS
LIN {X 0.079,Y -396.372,Z 1140.848,A 0.000,B 0.000,C 90.000,E1 8.681} C_DIS
LIN {X -0.103,Y -401.824,Z 1140.839,A 0.000,B 0.000,C 90.000,E1 6.947} C_DIS
LIN {X -0.171,Y -404.475,Z 1140.835,A 0.000,B 0.000,C 90.000,E1 6.258} C_DIS
LIN {X -0.174,Y -406.240,Z 1140.833,A 0.000,B 0.000,C 90.000,E1 5.910} C_DIS
LIN {X -0.194,Y -407.203,Z 1140.832,A 0.000,B 0.000,C 90.000,E1 5.739} C_DIS
LIN {X -0.213,Y -408.367,Z 1140.831,A 0.000,B 0.000,C 90.000,E1 5.568} C_DIS
LIN {X -0.037,Y -411.896,Z 1140.828,A 0.000,B 0.000,C 90.000,E1 5.106} C_DIS
LIN {X -0.053,Y -419.460,Z 1140.825,A 0.000,B 0.000,C 90.000,E1 4.531} C_DIS
LIN {X -0.151,Y -429.137,Z 1140.821,A 0.000,B 0.000,C 90.000,E1 3.841} C_DIS
LIN {X -0.017,Y -453.614,Z 1140.812,A 0.000,B 0.000,C 90.000,E1 2.121} C_DIS
LIN {X 0.134,Y -471.475,Z 1140.805,A 0.000,B 0.000,C 90.000,E1 0.917} C_DIS
LIN {X 0.042,Y -484.128,Z 1140.800,A 0.000,B 0.000,C 90.000,E1 0.057} C_DIS
LIN {X 0.219,Y -490.950,Z 1140.798,A 0.000,B 0.000,C 90.000,E1 359.542} C_DIS
LIN {X 0.096,Y -498.489,Z 1140.794,A 0.000,B 0.000,C 90.000,E1 358.969} C_DIS
LIN {X -0.125,Y -504.366,Z 1140.792,A 0.000,B 0.000,C 90.000,E1 358.511} C_DIS
LIN {X 0.030,Y -510.100,Z 1140.789,A 0.000,B 0.000,C 90.000,E1 357.993} C_DIS
LIN {X 0.218,Y -518.053,Z 1140.785,A 0.000,B 0.000,C 90.000,E1 357.192} C_DIS
LIN {X 0.168,Y -521.996,Z 1140.782,A 0.000,B 0.000,C 90.000,E1 356.788} C_DIS
LIN {X 0.170,Y -527.152,Z 1140.779,A 0.000,B 0.000,C 90.000,E1 356.216} C_DIS
LIN {X -0.104,Y -533.004,Z 1140.775,A 0.000,B 0.000,C 90.000,E1 355.527} C_DIS
LIN {X -0.091,Y -537.279,Z 1140.772,A 0.000,B 0.000,C 90.000,E1 354.951} C_DIS
LIN {X 0.226,Y -542.012,Z 1140.768,A 0.000,B 0.000,C 90.000,E1 354.204} C_DIS
LIN {X 0.047,Y -546.338,Z 1140.764,A 0.000,B 0.000,C 90.000,E1 353.514} C_DIS
LIN {X -0.035,Y -550.252,Z 1140.760,A 0.000,B 0.000,C 90.000,E1 352.818} C_DIS
LIN {X -0.151,Y -553.698,Z 1140.756,A 0.000,B 0.000,C 90.000,E1 352.129} C_DIS
LIN {X 0.090,Y -556.286,Z 1140.753,A 0.000,B 0.000,C 90.000,E1 351.546} C_DIS
LIN {X 0.105,Y -559.203,Z 1140.749,A 0.000,B 0.000,C 90.000,E1 350.849} C_DIS
LIN {X -0.106,Y -562.352,Z 1140.745,A 0.000,B 0.000,C 90.000,E1 350.038} C_DIS
LIN {X -0.187,Y -565.249,Z 1140.740,A 0.000,B 0.000,C 90.000,E1 349.218} C_DIS
LIN {X -0.174,Y -568.747,Z 1140.734,A 0.000,B 0.000,C 90.000,E1 348.117} C_DIS
LIN {X 0.124,Y -571.929,Z 1140.728,A 0.000,B 0.000,C 90.000,E1 346.992} C_DIS
LIN {X -0.213,Y -574.938,Z 1140.722,A 0.000,B 0.000,C 90.000,E1 345.936} C_DIS
LIN {X 0.186,Y -577.808,Z 1140.716,A 0.000,B 0.000,C 90.000,E1 344.810} C_DIS
LIN {X 0.106,Y -581.843,Z 1140.707,A 0.000,B 0.000,C 90.000,E1 343.196} C_DIS
LIN {X -0.117,Y -585.051,Z 1140.699,A 0.000,B 0.000,C 90.000,E1 341.873} C_DIS
LIN {X -0.292,Y -587.907,Z 1140.692,A 0.000,B 0.000,C 90.000,E1 340.550} C_DIS
LIN {X 0.223,Y -589.499,Z 1140.687,A 0.000,B 0.000,C 90.000,E1 339.699} C_DIS
LIN {X 0.088,Y -591.429,Z 1140.682,A 0.000,B 0.000,C 90.000,E1 338.646} C_DIS
LIN {X 0.090,Y -592.677,Z 1140.677,A 0.000,B 0.000,C 90.000,E1 337.847} C_DIS
LIN {X 0.001,Y -593.949,Z 1140.671,A 0.000,B 0.000,C 90.000,E1 336.794} C_DIS
LIN {X 0.017,Y -594.745,Z 1140.667,A 0.000,B 0.000,C 90.000,E1 335.997} C_DIS
LIN {X 0.188,Y -595.436,Z 1140.661,A 0.000,B 0.000,C 90.000,E1 334.921} C_DIS
LIN {X -0.077,Y -595.681,Z 1140.656,A 0.000,B 0.000,C 90.000,E1 334.152} C_DIS
LIN {X 0.194,Y -595.576,Z 1140.652,A 0.000,B 0.000,C 90.000,E1 333.332} C_DIS
LIN {X 0.115,Y -594.830,Z 1140.646,A 0.000,B 0.000,C 90.000,E1 332.281} C_DIS
LIN {X -0.064,Y -594.303,Z 1140.643,A 0.000,B 0.000,C 90.000,E1 331.769} C_DIS
LIN {X -0.152,Y -592.817,Z 1140.637,A 0.000,B 0.000,C 90.000,E1 330.717} C_DIS
LIN {X -0.350,Y -591.722,Z 1140.634,A 0.000,B 0.000,C 90.000,E1 330.205} C_DIS
LIN {X -0.260,Y -590.461,Z 1140.631,A 0.000,B 0.000,C 90.000,E1 329.665} C_DIS
LIN {X -0.290,Y -588.281,Z 1140.627,A 0.000,B 0.000,C 90.000,E1 328.869} C_DIS
LIN {X -0.036,Y -585.393,Z 1140.622,A 0.000,B 0.000,C 90.000,E1 328.043} C_DIS
LIN {X -0.052,Y -582.577,Z 1140.619,A 0.000,B 0.000,C 90.000,E1 327.375} C_DIS
LIN {X -0.102,Y -579.104,Z 1140.615,A 0.000,B 0.000,C 90.000,E1 326.707} C_DIS
LIN {X 0.133,Y -575.297,Z 1140.611,A 0.000,B 0.000,C 90.000,E1 326.008} C_DIS
LIN {X 0.103,Y -572.004,Z 1140.608,A 0.000,B 0.000,C 90.000,E1 325.468} C_DIS
LIN {X -0.191,Y -567.277,Z 1140.604,A 0.000,B 0.000,C 90.000,E1 324.815} C_DIS
LIN {X -0.280,Y -563.184,Z 1140.601,A 0.000,B 0.000,C 90.000,E1 324.276} C_DIS
LIN {X -0.070,Y -558.799,Z 1140.598,A 0.000,B 0.000,C 90.000,E1 323.703} C_DIS
LIN {X -0.102,Y -555.344,Z 1140.596,A 0.000,B 0.000,C 90.000,E1 323.290} C_DIS
LIN {X 0.085,Y -546.697,Z 1140.591,A 0.000,B 0.000,C 90.000,E1 322.316} C_DIS
LIN {X -0.143,Y -534.058,Z 1140.583,A 0.000,B 0.000,C 90.000,E1 320.964} C_DIS
LIN {X -0.047,Y -530.060,Z 1140.580,A 0.000,B 0.000,C 90.000,E1 320.436} C_DIS
LIN {X 0.028,Y -527.818,Z 1140.578,A 0.000,B 0.000,C 90.000,E1 320.070} C_DIS
LIN {X -0.120,Y -526.158,Z 1140.576,A 0.000,B 0.000,C 90.000,E1 319.747} C_DIS
LIN {X -0.152,Y -524.996,Z 1140.575,A 0.000,B 0.000,C 90.000,E1 319.461} C_DIS
LIN {X -0.217,Y -523.809,Z 1140.572,A 0.000,B 0.000,C 90.000,E1 319.013} C_DIS
LIN {X 0.032,Y -522.606,Z 1140.567,A 0.000,B 0.000,C 90.000,E1 318.119} C_DIS
LIN {X 0.123,Y -522.215,Z 1140.561,A 0.000,B 0.000,C 90.000,E1 316.944} C_DIS
LIN {X -0.004,Y -522.853,Z 1140.550,A 0.000,B 0.000,C 90.000,E1 314.919} C_DIS
LIN {X 0.023,Y -523.261,Z 1140.542,A 0.000,B 0.000,C 90.000,E1 313.461} C_DIS
LIN {X 0.029,Y -523.823,Z 1140.532,A 0.000,B 0.000,C 90.000,E1 311.714} C_DIS
LIN {X -0.046,Y -524.795,Z 1140.521,A 0.000,B 0.000,C 90.000,E1 309.688} C_DIS
LIN {X 0.025,Y -525.927,Z 1140.509,A 0.000,B 0.000,C 90.000,E1 307.649} C_DIS
LIN {X -0.161,Y -527.031,Z 1140.500,A 0.000,B 0.000,C 90.000,E1 305.931} C_DIS
LIN {X -0.201,Y -528.202,Z 1140.490,A 0.000,B 0.000,C 90.000,E1 304.199} C_DIS
LIN {X 0.232,Y -529.332,Z 1140.480,A 0.000,B 0.000,C 90.000,E1 302.418} C_DIS
LIN {X 0.107,Y -530.837,Z 1140.469,A 0.000,B 0.000,C 90.000,E1 300.413} C_DIS
LIN {X -0.126,Y -531.779,Z 1140.461,A 0.000,B 0.000,C 90.000,E1 298.999} C_DIS
LIN {X 0.184,Y -532.355,Z 1140.456,A 0.000,B 0.000,C 90.000,E1 298.103} C_DIS
LIN {X -0.067,Y -532.928,Z 1140.448,A 0.000,B 0.000,C 90.000,E1 296.693} C_DIS
LIN {X 0.113,Y -533.281,Z 1140.439,A 0.000,B 0.000,C 90.000,E1 294.951} C_DIS
LIN {X 0.128,Y -533.327,Z 1140.431,A 0.000,B 0.000,C 90.000,E1 293.515} C_DIS
LIN {X -0.150,Y -533.300,Z 1140.420,A 0.000,B 0.000,C 90.000,E1 291.535} C_DIS
LIN {X 0.166,Y -533.195,Z 1140.412,A 0.000,B 0.000,C 90.000,E1 290.066} C_DIS
LIN {X -0.201,Y -532.876,Z 1140.404,A 0.000,B 0.000,C 90.000,E1 288.671} C_DIS
LIN {X -0.102,Y -532.550,Z 1140.397,A 0.000,B 0.000,C 90.000,E1 287.511} C_DIS
LIN {X -0.145,Y -532.008,Z 1140.389,A 0.000,B 0.000,C 90.000,E1 286.079} C_DIS
LIN {X 0.143,Y -531.516,Z 1140.383,A 0.000,B 0.000,C 90.000,E1 284.898} C_DIS
LIN {X -0.088,Y -530.875,Z 1140.376,A 0.000,B 0.000,C 90.000,E1 283.772} C_DIS
LIN {X -0.191,Y -529.641,Z 1140.364,A 0.000,B 0.000,C 90.000,E1 281.478} C_DIS
LIN {X 0.006,Y -528.634,Z 1140.354,A 0.000,B 0.000,C 90.000,E1 279.726} C_DIS
LIN {X 0.033,Y -527.980,Z 1140.348,A 0.000,B 0.000,C 90.000,E1 278.568} C_DIS
LIN {X 0.004,Y -527.180,Z 1140.340,A 0.000,B 0.000,C 90.000,E1 277.125} C_DIS
LIN {X -0.068,Y -526.182,Z 1140.328,A 0.000,B 0.000,C 90.000,E1 275.106} C_DIS
LIN {X -0.224,Y -525.333,Z 1140.317,A 0.000,B 0.000,C 90.000,E1 273.094} C_DIS
LIN {X 0.098,Y -524.613,Z 1140.307,A 0.000,B 0.000,C 90.000,E1 271.318} C_DIS
LIN {X -0.125,Y -523.859,Z 1140.298,A 0.000,B 0.000,C 90.000,E1 269.599} C_DIS
LIN {X 0.129,Y -522.913,Z 1140.286,A 0.000,B 0.000,C 90.000,E1 267.535} C_DIS
LIN {X -0.092,Y -522.028,Z 1140.277,A 0.000,B 0.000,C 90.000,E1 265.812} C_DIS
LIN {X 0.243,Y -521.128,Z 1140.269,A 0.000,B 0.000,C 90.000,E1 264.318} C_DIS
LIN {X 0.107,Y -520.400,Z 1140.264,A 0.000,B 0.000,C 90.000,E1 263.457} C_DIS
LIN {X -0.079,Y -518.672,Z 1140.254,A 0.000,B 0.000,C 90.000,E1 261.724} C_DIS
LIN {X -0.249,Y -516.279,Z 1140.241,A 0.000,B 0.000,C 90.000,E1 259.398} C_DIS
LIN {X 0.133,Y -514.193,Z 1140.230,A 0.000,B 0.000,C 90.000,E1 257.297} C_DIS
LIN {X 0.150,Y -512.081,Z 1140.216,A 0.000,B 0.000,C 90.000,E1 254.936} C_DIS
LIN {X -0.160,Y -510.460,Z 1140.207,A 0.000,B 0.000,C 90.000,E1 253.196} C_DIS
LIN {X -0.015,Y -508.699,Z 1140.197,A 0.000,B 0.000,C 90.000,E1 251.402} C_DIS
LIN {X 0.116,Y -507.799,Z 1140.192,A 0.000,B 0.000,C 90.000,E1 250.496} C_DIS
LIN {X 0.135,Y -505.597,Z 1140.180,A 0.000,B 0.000,C 90.000,E1 248.411} C_DIS
LIN {X 0.199,Y -503.565,Z 1140.170,A 0.000,B 0.000,C 90.000,E1 246.613} C_DIS
LIN {X 0.057,Y -502.055,Z 1140.164,A 0.000,B 0.000,C 90.000,E1 245.433} C_DIS
LIN {X -0.004,Y -499.600,Z 1140.154,A 0.000,B 0.000,C 90.000,E1 243.640} C_DIS
LIN {X -0.161,Y -497.406,Z 1140.145,A 0.000,B 0.000,C 90.000,E1 242.153} C_DIS
LIN {X 0.313,Y -495.129,Z 1140.137,A 0.000,B 0.000,C 90.000,E1 240.589} C_DIS
LIN {X 0.144,Y -492.196,Z 1140.127,A 0.000,B 0.000,C 90.000,E1 238.791} C_DIS
LIN {X -0.262,Y -488.792,Z 1140.115,A 0.000,B 0.000,C 90.000,E1 236.707} C_DIS
LIN {X -0.057,Y -485.770,Z 1140.105,A 0.000,B 0.000,C 90.000,E1 234.848} C_DIS
LIN {X -0.043,Y -482.746,Z 1140.094,A 0.000,B 0.000,C 90.000,E1 233.004} C_DIS
LIN {X -0.186,Y -479.557,Z 1140.084,A 0.000,B 0.000,C 90.000,E1 231.170} C_DIS
LIN {X -0.196,Y -476.854,Z 1140.076,A 0.000,B 0.000,C 90.000,E1 229.622} C_DIS
LIN {X 0.140,Y -473.598,Z 1140.065,A 0.000,B 0.000,C 90.000,E1 227.715} C_DIS
LIN {X -0.208,Y -469.789,Z 1140.053,A 0.000,B 0.000,C 90.000,E1 225.567} C_DIS
LIN {X 0.029,Y -464.445,Z 1140.032,A 0.000,B 0.000,C 90.000,E1 221.757} C_DIS
LIN {X -0.032,Y -461.115,Z 1140.016,A 0.000,B 0.000,C 90.000,E1 218.910} C_DIS
LIN {X 0.223,Y -458.252,Z 1140.000,A 0.000,B 0.000,C 90.000,E1 216.011} C_DIS
LIN {X -0.017,Y -455.219,Z 1139.977,A 0.000,B 0.000,C 90.000,E1 211.878} C_DIS
LIN {X -0.038,Y -454.411,Z 1139.956,A 0.000,B 0.000,C 90.000,E1 208.025} C_DIS
LIN {X 0.002,Y -455.324,Z 1139.943,A 0.000,B 0.000,C 90.000,E1 205.771} C_DIS
LIN {X 0.198,Y -456.451,Z 1139.936,A 0.000,B 0.000,C 90.000,E1 204.463} C_DIS
LIN {X 0.002,Y -458.122,Z 1139.929,A 0.000,B 0.000,C 90.000,E1 203.206} C_DIS
LIN {X 0.086,Y -461.457,Z 1139.918,A 0.000,B 0.000,C 90.000,E1 201.280} C_DIS
LIN {X -0.146,Y -466.455,Z 1139.906,A 0.000,B 0.000,C 90.000,E1 199.087} C_DIS
LIN {X 0.057,Y -472.653,Z 1139.894,A 0.000,B 0.000,C 90.000,E1 196.858} C_DIS
LIN {X 0.142,Y -480.932,Z 1139.880,A 0.000,B 0.000,C 90.000,E1 194.356} C_DIS
LIN {X -0.100,Y -487.515,Z 1139.870,A 0.000,B 0.000,C 90.000,E1 192.535} C_DIS
LIN {X -0.198,Y -494.331,Z 1139.859,A 0.000,B 0.000,C 90.000,E1 190.715} C_DIS
LIN {X 0.162,Y -501.283,Z 1139.849,A 0.000,B 0.000,C 90.000,E1 188.859} C_DIS
LIN {X 0.127,Y -508.347,Z 1139.839,A 0.000,B 0.000,C 90.000,E1 187.068} C_DIS
LIN {X 0.244,Y -515.304,Z 1139.829,A 0.000,B 0.000,C 90.000,E1 185.277} C_DIS
LIN {X -0.102,Y -522.216,Z 1139.820,A 0.000,B 0.000,C 90.000,E1 183.555} C_DIS
LIN {X -0.260,Y -526.820,Z 1139.813,A 0.000,B 0.000,C 90.000,E1 182.407} C_DIS
LIN {X 0.146,Y -533.671,Z 1139.804,A 0.000,B 0.000,C 90.000,E1 180.630} C_DIS
LIN {X 0.163,Y -540.560,Z 1139.794,A 0.000,B 0.000,C 90.000,E1 178.912} C_DIS
LIN {X -0.242,Y -546.277,Z 1139.786,A 0.000,B 0.000,C 90.000,E1 177.535} C_DIS
LIN {X -0.002,Y -552.018,Z 1139.778,A 0.000,B 0.000,C 90.000,E1 176.102} C_DIS
LIN {X -0.054,Y -558.876,Z 1139.769,A 0.000,B 0.000,C 90.000,E1 174.432} C_DIS
LIN {X -0.107,Y -564.579,Z 1139.761,A 0.000,B 0.000,C 90.000,E1 173.053} C_DIS
LIN {X 0.081,Y -570.280,Z 1139.754,A 0.000,B 0.000,C 90.000,E1 171.659} C_DIS
LIN {X -0.075,Y -577.019,Z 1139.745,A 0.000,B 0.000,C 90.000,E1 170.038} C_DIS
LIN {X -0.232,Y -582.432,Z 1139.737,A 0.000,B 0.000,C 90.000,E1 168.701} C_DIS
LIN {X -0.102,Y -585.641,Z 1139.733,A 0.000,B 0.000,C 90.000,E1 167.881} C_DIS
LIN {X -0.256,Y -589.821,Z 1139.727,A 0.000,B 0.000,C 90.000,E1 166.825} C_DIS
LIN {X -0.213,Y -593.863,Z 1139.721,A 0.000,B 0.000,C 90.000,E1 165.755} C_DIS
LIN {X -0.104,Y -597.679,Z 1139.715,A 0.000,B 0.000,C 90.000,E1 164.685} C_DIS
LIN {X -0.223,Y -602.166,Z 1139.708,A 0.000,B 0.000,C 90.000,E1 163.378} C_DIS
LIN {X 0.210,Y -607.255,Z 1139.699,A 0.000,B 0.000,C 90.000,E1 161.764} C_DIS
LIN {X 0.105,Y -610.481,Z 1139.693,A 0.000,B 0.000,C 90.000,E1 160.732} C_DIS
LIN {X -0.002,Y -614.293,Z 1139.686,A 0.000,B 0.000,C 90.000,E1 159.444} C_DIS
LIN {X -0.043,Y -617.824,Z 1139.679,A 0.000,B 0.000,C 90.000,E1 158.156} C_DIS
LIN {X -0.044,Y -621.954,Z 1139.670,A 0.000,B 0.000,C 90.000,E1 156.613} C_DIS
LIN {X -0.281,Y -626.563,Z 1139.660,A 0.000,B 0.000,C 90.000,E1 154.845} C_DIS
LIN {X -0.186,Y -629.681,Z 1139.653,A 0.000,B 0.000,C 90.000,E1 153.563} C_DIS
LIN {X -0.036,Y -632.607,Z 1139.646,A 0.000,B 0.000,C 90.000,E1 152.281} C_DIS
LIN {X 0.150,Y -635.407,Z 1139.639,A 0.000,B 0.000,C 90.000,E1 151.001} C_DIS
LIN {X 0.129,Y -638.086,Z 1139.632,A 0.000,B 0.000,C 90.000,E1 149.744} C_DIS
LIN {X 0.150,Y -640.656,Z 1139.625,A 0.000,B 0.000,C 90.000,E1 148.486} C_DIS
LIN {X -0.050,Y -642.595,Z 1139.620,A 0.000,B 0.000,C 90.000,E1 147.502} C_DIS
LIN {X -0.092,Y -645.312,Z 1139.611,A 0.000,B 0.000,C 90.000,E1 146.008} C_DIS
LIN {X 0.271,Y -647.915,Z 1139.603,A 0.000,B 0.000,C 90.000,E1 144.482} C_DIS
LIN {X 0.150,Y -650.422,Z 1139.595,A 0.000,B 0.000,C 90.000,E1 143.004} C_DIS
LIN {X -0.112,Y -653.386,Z 1139.585,A 0.000,B 0.000,C 90.000,E1 141.295} C_DIS
LIN {X 0.131,Y -657.535,Z 1139.573,A 0.000,B 0.000,C 90.000,E1 139.057} C_DIS
LIN {X 0.026,Y -660.944,Z 1139.563,A 0.000,B 0.000,C 90.000,E1 137.349} C_DIS
LIN {X -0.096,Y -664.838,Z 1139.552,A 0.000,B 0.000,C 90.000,E1 135.405} C_DIS
LIN {X -0.098,Y -669.679,Z 1139.540,A 0.000,B 0.000,C 90.000,E1 133.218} C_DIS
LIN {X 0.037,Y -674.292,Z 1139.529,A 0.000,B 0.000,C 90.000,E1 131.272} C_DIS
LIN {X 0.329,Y -678.352,Z 1139.520,A 0.000,B 0.000,C 90.000,E1 129.564} C_DIS
LIN {X 0.300,Y -682.668,Z 1139.511,A 0.000,B 0.000,C 90.000,E1 127.890} C_DIS
LIN {X -0.219,Y -686.265,Z 1139.503,A 0.000,B 0.000,C 90.000,E1 126.503} C_DIS
LIN {X -0.164,Y -689.230,Z 1139.496,A 0.000,B 0.000,C 90.000,E1 125.311} C_DIS
LIN {X 0.156,Y -692.706,Z 1139.488,A 0.000,B 0.000,C 90.000,E1 123.865} C_DIS
LIN {X 0.312,Y -695.490,Z 1139.482,A 0.000,B 0.000,C 90.000,E1 122.673} C_DIS
LIN {X 0.100,Y -697.566,Z 1139.476,A 0.000,B 0.000,C 90.000,E1 121.750} C_DIS
LIN {X 0.028,Y -698.912,Z 1139.473,A 0.000,B 0.000,C 90.000,E1 121.052} C_DIS
LIN {X 0.130,Y -700.949,Z 1139.466,A 0.000,B 0.000,C 90.000,E1 119.873} C_DIS
LIN {X 0.273,Y -703.037,Z 1139.460,A 0.000,B 0.000,C 90.000,E1 118.693} C_DIS
LIN {X -0.123,Y -704.209,Z 1139.456,A 0.000,B 0.000,C 90.000,E1 118.025} C_DIS
LIN {X -0.216,Y -705.099,Z 1139.452,A 0.000,B 0.000,C 90.000,E1 117.334} C_DIS
LIN {X -0.265,Y -705.574,Z 1139.449,A 0.000,B 0.000,C 90.000,E1 116.873} C_DIS
LIN {X 0.250,Y -706.242,Z 1139.443,A 0.000,B 0.000,C 90.000,E1 115.668} C_DIS
LIN {X 0.192,Y -706.324,Z 1139.439,A 0.000,B 0.000,C 90.000,E1 114.975} C_DIS
LIN {X 0.136,Y -706.163,Z 1139.436,A 0.000,B 0.000,C 90.000,E1 114.515} C_DIS
LIN {X -0.216,Y -705.324,Z 1139.434,A 0.000,B 0.000,C 90.000,E1 114.079} C_DIS
LIN {X 0.072,Y -704.676,Z 1139.432,A 0.000,B 0.000,C 90.000,E1 113.823} C_DIS
LIN {X -0.287,Y -702.726,Z 1139.430,A 0.000,B 0.000,C 90.000,E1 113.387} C_DIS
LIN {X -0.148,Y -702.051,Z 1139.429,A 0.000,B 0.000,C 90.000,E1 113.259} C_DIS
LIN {X -0.012,Y -698.805,Z 1139.427,A 0.000,B 0.000,C 90.000,E1 112.898} C_DIS
LIN {X 0.252,Y -696.402,Z 1139.426,A 0.000,B 0.000,C 90.000,E1 112.642} C_DIS
LIN {X 0.425,Y -694.528,Z 1139.425,A 0.000,B 0.000,C 90.000,E1 112.514} C_DIS
LIN {X -0.065,Y -686.170,Z 1139.424,A 0.000,B 0.000,C 90.000,E1 112.259} C_DIS
LIN {X 0.214,Y -684.938,Z 1139.423,A 0.000,B 0.000,C 90.000,E1 112.206} C_DIS
LIN {X -0.134,Y -676.756,Z 1139.423,A 0.000,B 0.000,C 90.000,E1 112.153} C_DIS
LIN {X -0.167,Y -603.329,Z 1139.423,A 0.000,B 0.000,C 90.000,E1 112.153} C_DIS
LIN {X 0.201,Y -599.982,Z 1139.422,A 0.000,B 0.000,C 90.000,E1 111.897} C_DIS
LIN {X 0.234,Y -595.333,Z 1139.420,A 0.000,B 0.000,C 90.000,E1 111.535} C_DIS
LIN {X 0.013,Y -582.598,Z 1139.414,A 0.000,B 0.000,C 90.000,E1 110.429} C_DIS
LIN {X 0.115,Y -575.654,Z 1139.410,A 0.000,B 0.000,C 90.000,E1 109.812} C_DIS
LIN {X -0.208,Y -568.235,Z 1139.407,A 0.000,B 0.000,C 90.000,E1 109.268} C_DIS
LIN {X 0.005,Y -560.037,Z 1139.404,A 0.000,B 0.000,C 90.000,E1 108.725} C_DIS
LIN {X 0.303,Y -555.561,Z 1139.403,A 0.000,B 0.000,C 90.000,E1 108.417} C_DIS
LIN {X 0.234,Y -550.911,Z 1139.401,A 0.000,B 0.000,C 90.000,E1 108.055} C_DIS
LIN {X 0.201,Y -549.784,Z 1139.399,A 0.000,B 0.000,C 90.000,E1 107.873} C_DIS
LIN {X 0.158,Y -549.773,Z 1139.399,A 0.000,B 0.000,C 90.000,E1 107.873} C_DIS
LIN {X 0.036,Y -549.537,Z 1139.397,A 0.000,B 0.000,C 90.000,E1 107.457} C_DIS
LIN {X -0.186,Y -550.973,Z 1139.385,A 0.000,B 0.000,C 90.000,E1 105.245} C_DIS
LIN {X 0.087,Y -552.285,Z 1139.375,A 0.000,B 0.000,C 90.000,E1 103.536} C_DIS
LIN {X -0.152,Y -553.742,Z 1139.366,A 0.000,B 0.000,C 90.000,E1 101.883} C_DIS
LIN {X 0.082,Y -555.461,Z 1139.355,A 0.000,B 0.000,C 90.000,E1 99.905} C_DIS
LIN {X -0.035,Y -556.525,Z 1139.349,A 0.000,B 0.000,C 90.000,E1 98.803} C_DIS
LIN {X 0.054,Y -557.948,Z 1139.340,A 0.000,B 0.000,C 90.000,E1 97.125} C_DIS
LIN {X 0.110,Y -559.385,Z 1139.330,A 0.000,B 0.000,C 90.000,E1 95.454} C_DIS
LIN {X 0.188,Y -560.737,Z 1139.321,A 0.000,B 0.000,C 90.000,E1 93.784} C_DIS
LIN {X 0.219,Y -561.983,Z 1139.312,A 0.000,B 0.000,C 90.000,E1 92.121} C_DIS
LIN {X 0.174,Y -562.961,Z 1139.304,A 0.000,B 0.000,C 90.000,E1 90.745} C_DIS
LIN {X 0.134,Y -563.880,Z 1139.297,A 0.000,B 0.000,C 90.000,E1 89.370} C_DIS
LIN {X -0.224,Y -565.030,Z 1139.286,A 0.000,B 0.000,C 90.000,E1 87.478} C_DIS
LIN {X -0.073,Y -565.916,Z 1139.277,A 0.000,B 0.000,C 90.000,E1 85.812} C_DIS
LIN {X -0.167,Y -566.472,Z 1139.271,A 0.000,B 0.000,C 90.000,E1 84.723} C_DIS
LIN {X 0.058,Y -567.240,Z 1139.261,A 0.000,B 0.000,C 90.000,E1 83.053} C_DIS
LIN {X -0.195,Y -568.024,Z 1139.252,A 0.000,B 0.000,C 90.000,E1 81.432} C_DIS
LIN {X 0.040,Y -568.642,Z 1139.245,A 0.000,B 0.000,C 90.000,E1 80.038} C_DIS
LIN {X -0.285,Y -569.667,Z 1139.233,A 0.000,B 0.000,C 90.000,E1 77.881} C_DIS
LIN {X 0.211,Y -570.312,Z 1139.225,A 0.000,B 0.000,C 90.000,E1 76.464} C_DIS
LIN {X 0.173,Y -570.948,Z 1139.217,A 0.000,B 0.000,C 90.000,E1 75.102} C_DIS
LIN {X 0.145,Y -571.725,Z 1139.210,A 0.000,B 0.000,C 90.000,E1 73.740} C_DIS
LIN {X -0.084,Y -572.788,Z 1139.201,A 0.000,B 0.000,C 90.000,E1 72.127} C_DIS
LIN {X 0.244,Y -574.256,Z 1139.190,A 0.000,B 0.000,C 90.000,E1 70.188} C_DIS
LIN {X 0.108,Y -576.147,Z 1139.178,A 0.000,B 0.000,C 90.000,E1 68.028} C_DIS
LIN {X 0.025,Y -577.713,Z 1139.169,A 0.000,B 0.000,C 90.000,E1 66.410} C_DIS
LIN {X -0.179,Y -579.435,Z 1139.158,A 0.000,B 0.000,C 90.000,E1 64.537} C_DIS
LIN {X 0.147,Y -581.086,Z 1139.148,A 0.000,B 0.000,C 90.000,E1 62.615} C_DIS
LIN {X 0.123,Y -582.402,Z 1139.139,A 0.000,B 0.000,C 90.000,E1 61.001} C_DIS
LIN {X 0.030,Y -583.360,Z 1139.132,A 0.000,B 0.000,C 90.000,E1 59.665} C_DIS
LIN {X 0.095,Y -584.164,Z 1139.126,A 0.000,B 0.000,C 90.000,E1 58.584} C_DIS
LIN {X -0.101,Y -585.111,Z 1139.117,A 0.000,B 0.000,C 90.000,E1 56.993} C_DIS
LIN {X 0.051,Y -586.217,Z 1139.106,A 0.000,B 0.000,C 90.000,E1 55.102} C_DIS
LIN {X 0.041,Y -587.114,Z 1139.097,A 0.000,B 0.000,C 90.000,E1 53.497} C_DIS
LIN {X -0.077,Y -587.888,Z 1139.088,A 0.000,B 0.000,C 90.000,E1 51.904} C_DIS
LIN {X -0.008,Y -588.459,Z 1139.081,A 0.000,B 0.000,C 90.000,E1 50.561} C_DIS
LIN {X 0.132,Y -588.732,Z 1139.077,A 0.000,B 0.000,C 90.000,E1 49.747} C_DIS
LIN {X 0.212,Y -588.865,Z 1139.069,A 0.000,B 0.000,C 90.000,E1 48.405} C_DIS
LIN {X -0.002,Y -588.787,Z 1139.060,A 0.000,B 0.000,C 90.000,E1 46.824} C_DIS
LIN {X 0.277,Y -588.606,Z 1139.054,A 0.000,B 0.000,C 90.000,E1 45.729} C_DIS
LIN {X 0.130,Y -588.246,Z 1139.048,A 0.000,B 0.000,C 90.000,E1 44.676} C_DIS
LIN {X 0.223,Y -587.820,Z 1139.044,A 0.000,B 0.000,C 90.000,E1 43.866} C_DIS
LIN {X 0.055,Y -587.192,Z 1139.038,A 0.000,B 0.000,C 90.000,E1 42.813} C_DIS
LIN {X 0.164,Y -586.551,Z 1139.033,A 0.000,B 0.000,C 90.000,E1 42.000} C_DIS
LIN {X 0.019,Y -585.365,Z 1139.027,A 0.000,B 0.000,C 90.000,E1 40.943} C_DIS
LIN {X 0.044,Y -583.706,Z 1139.020,A 0.000,B 0.000,C 90.000,E1 39.600} C_DIS
LIN {X -0.141,Y -582.217,Z 1139.014,A 0.000,B 0.000,C 90.000,E1 38.543} C_DIS
LIN {X 0.102,Y -580.439,Z 1139.008,A 0.000,B 0.000,C 90.000,E1 37.443} C_DIS
LIN {X -0.035,Y -578.328,Z 1139.002,A 0.000,B 0.000,C 90.000,E1 36.377} C_DIS
LIN {X -0.357,Y -576.348,Z 1138.998,A 0.000,B 0.000,C 90.000,E1 35.598} C_DIS
LIN {X 0.101,Y -574.125,Z 1138.993,A 0.000,B 0.000,C 90.000,E1 34.739} C_DIS
LIN {X 0.203,Y -571.606,Z 1138.989,A 0.000,B 0.000,C 90.000,E1 33.913} C_DIS
LIN {X 0.153,Y -569.678,Z 1138.986,A 0.000,B 0.000,C 90.000,E1 33.372} C_DIS
LIN {X 0.211,Y -566.561,Z 1138.981,A 0.000,B 0.000,C 90.000,E1 32.546} C_DIS
LIN {X -0.067,Y -563.085,Z 1138.976,A 0.000,B 0.000,C 90.000,E1 31.750} C_DIS
LIN {X 0.015,Y -559.816,Z 1138.973,A 0.000,B 0.000,C 90.000,E1 31.052} C_DIS
LIN {X 0.036,Y -554.835,Z 1138.967,A 0.000,B 0.000,C 90.000,E1 30.079} C_DIS
LIN {X 0.155,Y -548.528,Z 1138.961,A 0.000,B 0.000,C 90.000,E1 28.949} C_DIS
LIN {X 0.041,Y -542.315,Z 1138.955,A 0.000,B 0.000,C 90.000,E1 27.975} C_DIS
LIN {X 0.122,Y -537.478,Z 1138.952,A 0.000,B 0.000,C 90.000,E1 27.257} C_DIS
LIN {X 0.055,Y -533.304,Z 1138.948,A 0.000,B 0.000,C 90.000,E1 26.693} C_DIS
LIN {X -0.251,Y -525.355,Z 1138.943,A 0.000,B 0.000,C 90.000,E1 25.720} C_DIS
LIN {X -0.147,Y -516.531,Z 1138.937,A 0.000,B 0.000,C 90.000,E1 24.695} C_DIS
LIN {X 0.108,Y -510.091,Z 1138.933,A 0.000,B 0.000,C 90.000,E1 23.951} C_DIS
LIN {X 0.184,Y -506.089,Z 1138.931,A 0.000,B 0.000,C 90.000,E1 23.515} C_DIS
LIN {X 0.092,Y -494.811,Z 1138.925,A 0.000,B 0.000,C 90.000,E1 22.408} C_DIS
LIN {X 0.157,Y -484.675,Z 1138.919,A 0.000,B 0.000,C 90.000,E1 21.461} C_DIS
LIN {X 0.209,Y -477.373,Z 1138.916,A 0.000,B 0.000,C 90.000,E1 20.791} C_DIS
LIN {X 0.106,Y -467.053,Z 1138.911,A 0.000,B 0.000,C 90.000,E1 19.885} C_DIS
LIN {X -0.064,Y -449.255,Z 1138.902,A 0.000,B 0.000,C 90.000,E1 18.308} C_DIS
LIN {X 0.007,Y -431.915,Z 1138.892,A 0.000,B 0.000,C 90.000,E1 16.622} C_DIS
LIN {X 0.211,Y -419.354,Z 1138.885,A 0.000,B 0.000,C 90.000,E1 15.245} C_DIS
LIN {X 0.157,Y -408.382,Z 1138.878,A 0.000,B 0.000,C 90.000,E1 13.953} C_DIS
LIN {X 0.143,Y -402.146,Z 1138.873,A 0.000,B 0.000,C 90.000,E1 13.119} C_DIS
LIN {X -0.171,Y -398.650,Z 1138.870,A 0.000,B 0.000,C 90.000,E1 12.647} C_DIS
LIN {X 0.191,Y -395.260,Z 1138.867,A 0.000,B 0.000,C 90.000,E1 12.007} C_DIS
LIN {X 0.181,Y -393.182,Z 1138.864,A 0.000,B 0.000,C 90.000,E1 11.478} C_DIS
LIN {X 0.158,Y -392.214,Z 1138.861,A 0.000,B 0.000,C 90.000,E1 10.950} C_DIS
LIN {X 0.057,Y -392.502,Z 1138.858,A 0.000,B 0.000,C 90.000,E1 10.433} C_DIS
LIN {X 0.173,Y -393.138,Z 1138.856,A 0.000,B 0.000,C 90.000,E1 10.018} C_DIS
LIN {X 0.130,Y -393.819,Z 1138.854,A 0.000,B 0.000,C 90.000,E1 9.670} C_DIS
LIN {X -0.017,Y -397.617,Z 1138.846,A 0.000,B 0.000,C 90.000,E1 8.276} C_DIS
LIN {X -0.192,Y -402.630,Z 1138.837,A 0.000,B 0.000,C 90.000,E1 6.720} C_DIS
LIN {X 0.195,Y -405.417,Z 1138.833,A 0.000,B 0.000,C 90.000,E1 5.967} C_DIS
LIN {X -0.127,Y -407.199,Z 1138.832,A 0.000,B 0.000,C 90.000,E1 5.682} C_DIS
LIN {X -0.190,Y -409.759,Z 1138.830,A 0.000,B 0.000,C 90.000,E1 5.334} C_DIS
LIN {X 0.146,Y -411.695,Z 1138.828,A 0.000,B 0.000,C 90.000,E1 5.049} C_DIS
LIN {X -0.014,Y -416.998,Z 1138.826,A 0.000,B 0.000,C 90.000,E1 4.645} C_DIS
LIN {X -0.009,Y -426.562,Z 1138.822,A 0.000,B 0.000,C 90.000,E1 3.955} C_DIS
LIN {X 0.106,Y -449.238,Z 1138.813,A 0.000,B 0.000,C 90.000,E1 2.350} C_DIS
LIN {X 0.091,Y -463.866,Z 1138.808,A 0.000,B 0.000,C 90.000,E1 1.375} C_DIS
LIN {X -0.044,Y -471.976,Z 1138.805,A 0.000,B 0.000,C 90.000,E1 0.859} C_DIS
LIN {X 0.000,Y -484.445,Z 1138.800,A 0.000,B 0.000,C 90.000,E1 360.000} C_DIS
LIN {X 0.225,Y -491.966,Z 1138.797,A 0.000,B 0.000,C 90.000,E1 359.427} C_DIS
LIN {X 0.164,Y -497.972,Z 1138.794,A 0.000,B 0.000,C 90.000,E1 358.969} C_DIS
LIN {X -0.001,Y -503.854,Z 1138.792,A 0.000,B 0.000,C 90.000,E1 358.511} C_DIS
LIN {X 0.159,Y -509.630,Z 1138.789,A 0.000,B 0.000,C 90.000,E1 357.993} C_DIS
LIN {X 0.123,Y -516.280,Z 1138.786,A 0.000,B 0.000,C 90.000,E1 357.364} C_DIS
LIN {X -0.120,Y -521.610,Z 1138.782,A 0.000,B 0.000,C 90.000,E1 356.846} C_DIS
LIN {X 0.195,Y -527.956,Z 1138.779,A 0.000,B 0.000,C 90.000,E1 356.102} C_DIS
LIN {X 0.126,Y -533.626,Z 1138.775,A 0.000,B 0.000,C 90.000,E1 355.412} C_DIS
LIN {X 0.145,Y -537.879,Z 1138.771,A 0.000,B 0.000,C 90.000,E1 354.837} C_DIS
LIN {X -0.070,Y -542.585,Z 1138.767,A 0.000,B 0.000,C 90.000,E1 354.147} C_DIS
LIN {X 0.014,Y -546.104,Z 1138.764,A 0.000,B 0.000,C 90.000,E1 353.571} C_DIS
LIN {X -0.070,Y -550.063,Z 1138.760,A 0.000,B 0.000,C 90.000,E1 352.875} C_DIS
LIN {X -0.185,Y -553.615,Z 1138.757,A 0.000,B 0.000,C 90.000,E1 352.186} C_DIS
LIN {X 0.055,Y -556.255,Z 1138.753,A 0.000,B 0.000,C 90.000,E1 351.602} C_DIS
LIN {X 0.071,Y -559.195,Z 1138.750,A 0.000,B 0.000,C 90.000,E1 350.905} C_DIS
LIN {X -0.140,Y -562.384,Z 1138.745,A 0.000,B 0.000,C 90.000,E1 350.095} C_DIS
LIN {X -0.220,Y -565.317,Z 1138.740,A 0.000,B 0.000,C 90.000,E1 349.275} C_DIS
LIN {X -0.203,Y -568.869,Z 1138.734,A 0.000,B 0.000,C 90.000,E1 348.173} C_DIS
LIN {X 0.161,Y -572.877,Z 1138.727,A 0.000,B 0.000,C 90.000,E1 346.769} C_DIS
LIN {X -0.033,Y -575.866,Z 1138.721,A 0.000,B 0.000,C 90.000,E1 345.700} C_DIS
LIN {X -0.178,Y -578.698,Z 1138.715,A 0.000,B 0.000,C 90.000,E1 344.629} C_DIS
LIN {X -0.068,Y -582.096,Z 1138.707,A 0.000,B 0.000,C 90.000,E1 343.268} C_DIS
LIN {X -0.296,Y -585.337,Z 1138.700,A 0.000,B 0.000,C 90.000,E1 341.945} C_DIS
LIN {X 0.189,Y -587.121,Z 1138.695,A 0.000,B 0.000,C 90.000,E1 341.094} C_DIS
LIN {X 0.242,Y -589.870,Z 1138.688,A 0.000,B 0.000,C 90.000,E1 339.752} C_DIS
LIN {X -0.211,Y -592.280,Z 1138.680,A 0.000,B 0.000,C 90.000,E1 338.465} C_DIS
LIN {X -0.203,Y -593.444,Z 1138.676,A 0.000,B 0.000,C 90.000,E1 337.667} C_DIS
LIN {X -0.285,Y -594.723,Z 1138.670,A 0.000,B 0.000,C 90.000,E1 336.613} C_DIS
LIN {X -0.021,Y -595.454,Z 1138.666,A 0.000,B 0.000,C 90.000,E1 335.793} C_DIS
LIN {X 0.168,Y -596.120,Z 1138.660,A 0.000,B 0.000,C 90.000,E1 334.717} C_DIS
LIN {X -0.086,Y -596.312,Z 1138.655,A 0.000,B 0.000,C 90.000,E1 333.948} C_DIS
LIN {X 0.280,Y -596.282,Z 1138.652,A 0.000,B 0.000,C 90.000,E1 333.384} C_DIS
LIN {X 0.025,Y -595.799,Z 1138.648,A 0.000,B 0.000,C 90.000,E1 332.615} C_DIS
LIN {X 0.043,Y -595.125,Z 1138.644,A 0.000,B 0.000,C 90.000,E1 331.820} C_DIS
LIN {X -0.225,Y -594.080,Z 1138.639,A 0.000,B 0.000,C 90.000,E1 331.051} C_DIS
LIN {X -0.122,Y -593.279,Z 1138.636,A 0.000,B 0.000,C 90.000,E1 330.511} C_DIS
LIN {X -0.120,Y -591.536,Z 1138.632,A 0.000,B 0.000,C 90.000,E1 329.715} C_DIS
LIN {X -0.134,Y -589.430,Z 1138.627,A 0.000,B 0.000,C 90.000,E1 328.918} C_DIS
LIN {X -0.175,Y -586.690,Z 1138.623,A 0.000,B 0.000,C 90.000,E1 328.122} C_DIS
LIN {X -0.249,Y -583.389,Z 1138.618,A 0.000,B 0.000,C 90.000,E1 327.327} C_DIS
LIN {X -0.051,Y -579.246,Z 1138.614,A 0.000,B 0.000,C 90.000,E1 326.501} C_DIS
LIN {X -0.053,Y -576.218,Z 1138.611,A 0.000,B 0.000,C 90.000,E1 325.960} C_DIS
LIN {X 0.154,Y -572.082,Z 1138.607,A 0.000,B 0.000,C 90.000,E1 325.261} C_DIS
LIN {X -0.041,Y -568.394,Z 1138.604,A 0.000,B 0.000,C 90.000,E1 324.736} C_DIS
LIN {X 0.102,Y -563.318,Z 1138.600,A 0.000,B 0.000,C 90.000,E1 324.036} C_DIS
LIN {X 0.097,Y -560.133,Z 1138.598,A 0.000,B 0.000,C 90.000,E1 323.623} C_DIS
LIN {X 0.282,Y -555.462,Z 1138.595,A 0.000,B 0.000,C 90.000,E1 323.050} C_DIS
LIN {X -0.321,Y -550.519,Z 1138.592,A 0.000,B 0.000,C 90.000,E1 322.557} C_DIS
LIN {X -0.075,Y -536.675,Z 1138.583,A 0.000,B 0.000,C 90.000,E1 321.009} C_DIS
LIN {X -0.249,Y -532.452,Z 1138.581,A 0.000,B 0.000,C 90.000,E1 320.517} C_DIS
LIN {X -0.081,Y -531.339,Z 1138.580,A 0.000,B 0.000,C 90.000,E1 320.356} C_DIS
LIN {X 0.072,Y -528.567,Z 1138.577,A 0.000,B 0.000,C 90.000,E1 319.908} C_DIS
LIN {X 0.017,Y -525.925,Z 1138.574,A 0.000,B 0.000,C 90.000,E1 319.337} C_DIS
LIN {X 0.223,Y -524.188,Z 1138.571,A 0.000,B 0.000,C 90.000,E1 318.690} C_DIS
LIN {X -0.109,Y -523.118,Z 1138.567,A 0.000,B 0.000,C 90.000,E1 318.000} C_DIS
LIN {X 0.083,Y -522.645,Z 1138.562,A 0.000,B 0.000,C 90.000,E1 317.106} C_DIS
LIN {X 0.265,Y -523.164,Z 1138.549,A 0.000,B 0.000,C 90.000,E1 314.757} C_DIS
LIN {X -0.006,Y -523.450,Z 1138.542,A 0.000,B 0.000,C 90.000,E1 313.623} C_DIS
LIN {X -0.133,Y -524.168,Z 1138.529,A 0.000,B 0.000,C 90.000,E1 311.310} C_DIS
LIN {X -0.140,Y -525.178,Z 1138.518,A 0.000,B 0.000,C 90.000,E1 309.277} C_DIS
LIN {X -0.077,Y -526.575,Z 1138.505,A 0.000,B 0.000,C 90.000,E1 306.950} C_DIS
LIN {X 0.159,Y -527.902,Z 1138.494,A 0.000,B 0.000,C 90.000,E1 304.898} C_DIS
LIN {X 0.145,Y -529.066,Z 1138.484,A 0.000,B 0.000,C 90.000,E1 303.166} C_DIS
LIN {X -0.046,Y -530.945,Z 1138.470,A 0.000,B 0.000,C 90.000,E1 300.590} C_DIS
LIN {X -0.079,Y -531.917,Z 1138.462,A 0.000,B 0.000,C 90.000,E1 299.155} C_DIS
LIN {X 0.200,Y -532.653,Z 1138.456,A 0.000,B 0.000,C 90.000,E1 297.975} C_DIS
LIN {X -0.045,Y -533.237,Z 1138.448,A 0.000,B 0.000,C 90.000,E1 296.565} C_DIS
LIN {X -0.281,Y -533.533,Z 1138.440,A 0.000,B 0.000,C 90.000,E1 295.155} C_DIS
LIN {X -0.040,Y -533.610,Z 1138.432,A 0.000,B 0.000,C 90.000,E1 293.695} C_DIS
LIN {X -0.223,Y -533.576,Z 1138.424,A 0.000,B 0.000,C 90.000,E1 292.280} C_DIS
LIN {X 0.089,Y -533.557,Z 1138.417,A 0.000,B 0.000,C 90.000,E1 291.099} C_DIS
LIN {X -0.096,Y -533.387,Z 1138.409,A 0.000,B 0.000,C 90.000,E1 289.685} C_DIS
LIN {X 0.062,Y -533.025,Z 1138.400,A 0.000,B 0.000,C 90.000,E1 287.946} C_DIS
LIN {X -0.105,Y -532.314,Z 1138.389,A 0.000,B 0.000,C 90.000,E1 285.953} C_DIS
LIN {X 0.220,Y -531.624,Z 1138.381,A 0.000,B 0.000,C 90.000,E1 284.481} C_DIS
LIN {X 0.065,Y -530.672,Z 1138.371,A 0.000,B 0.000,C 90.000,E1 282.771} C_DIS
LIN {X -0.224,Y -529.788,Z 1138.361,A 0.000,B 0.000,C 90.000,E1 281.074} C_DIS
LIN {X 0.008,Y -528.618,Z 1138.350,A 0.000,B 0.000,C 90.000,E1 279.029} C_DIS
LIN {X 0.008,Y -527.612,Z 1138.341,A 0.000,B 0.000,C 90.000,E1 277.296} C_DIS
LIN {X -0.069,Y -526.778,Z 1138.331,A 0.000,B 0.000,C 90.000,E1 275.568} C_DIS
LIN {X -0.166,Y -526.113,Z 1138.323,A 0.000,B 0.000,C 90.000,E1 274.131} C_DIS
LIN {X 0.245,Y -525.508,Z 1138.315,A 0.000,B 0.000,C 90.000,E1 272.636} C_DIS
LIN {X 0.088,Y -524.937,Z 1138.307,A 0.000,B 0.000,C 90.000,E1 271.203} C_DIS
LIN {X -0.129,Y -524.186,Z 1138.297,A 0.000,B 0.000,C 90.000,E1 269.484} C_DIS
LIN {X 0.133,Y -523.229,Z 1138.286,A 0.000,B 0.000,C 90.000,E1 267.421} C_DIS
LIN {X -0.082,Y -522.297,Z 1138.276,A 0.000,B 0.000,C 90.000,E1 265.698} C_DIS
LIN {X -0.206,Y -521.636,Z 1138.270,A 0.000,B 0.000,C 90.000,E1 264.546} C_DIS
LIN {X 0.180,Y -520.650,Z 1138.263,A 0.000,B 0.000,C 90.000,E1 263.337} C_DIS
LIN {X 0.011,Y -518.939,Z 1138.253,A 0.000,B 0.000,C 90.000,E1 261.602} C_DIS
LIN {X -0.137,Y -516.543,Z 1138.240,A 0.000,B 0.000,C 90.000,E1 259.275} C_DIS
LIN {X 0.239,Y -514.199,Z 1138.227,A 0.000,B 0.000,C 90.000,E1 256.881} C_DIS
LIN {X -0.233,Y -512.132,Z 1138.214,A 0.000,B 0.000,C 90.000,E1 254.574} C_DIS
LIN {X -0.151,Y -510.733,Z 1138.206,A 0.000,B 0.000,C 90.000,E1 253.087} C_DIS
LIN {X 0.255,Y -508.657,Z 1138.194,A 0.000,B 0.000,C 90.000,E1 250.967} C_DIS
LIN {X -0.163,Y -507.351,Z 1138.188,A 0.000,B 0.000,C 90.000,E1 249.826} C_DIS
LIN {X -0.153,Y -505.778,Z 1138.180,A 0.000,B 0.000,C 90.000,E1 248.337} C_DIS
LIN {X -0.162,Y -504.099,Z 1138.171,A 0.000,B 0.000,C 90.000,E1 246.847} C_DIS
LIN {X -0.208,Y -502.215,Z 1138.163,A 0.000,B 0.000,C 90.000,E1 245.357} C_DIS
LIN {X 0.190,Y -499.744,Z 1138.153,A 0.000,B 0.000,C 90.000,E1 243.512} C_DIS
LIN {X 0.034,Y -497.547,Z 1138.145,A 0.000,B 0.000,C 90.000,E1 242.025} C_DIS
LIN {X 0.105,Y -494.729,Z 1138.135,A 0.000,B 0.000,C 90.000,E1 240.205} C_DIS
LIN {X -0.083,Y -492.234,Z 1138.126,A 0.000,B 0.000,C 90.000,E1 238.712} C_DIS
LIN {X -0.049,Y -489.326,Z 1138.116,A 0.000,B 0.000,C 90.000,E1 236.882} C_DIS
LIN {X 0.071,Y -486.814,Z 1138.108,A 0.000,B 0.000,C 90.000,E1 235.341} C_DIS
LIN {X 0.107,Y -483.775,Z 1138.097,A 0.000,B 0.000,C 90.000,E1 233.497} C_DIS
LIN {X -0.123,Y -481.126,Z 1138.089,A 0.000,B 0.000,C 90.000,E1 231.984} C_DIS
LIN {X 0.092,Y -478.993,Z 1138.082,A 0.000,B 0.000,C 90.000,E1 230.723} C_DIS
LIN {X -0.041,Y -475.141,Z 1138.070,A 0.000,B 0.000,C 90.000,E1 228.566} C_DIS
LIN {X 0.036,Y -472.981,Z 1138.063,A 0.000,B 0.000,C 90.000,E1 227.310} C_DIS
LIN {X -0.082,Y -467.757,Z 1138.046,A 0.000,B 0.000,C 90.000,E1 224.190} C_DIS
LIN {X -0.173,Y -464.278,Z 1138.031,A 0.000,B 0.000,C 90.000,E1 221.676} C_DIS
LIN {X -0.241,Y -460.863,Z 1138.016,A 0.000,B 0.000,C 90.000,E1 218.830} C_DIS
LIN {X -0.005,Y -458.251,Z 1138.001,A 0.000,B 0.000,C 90.000,E1 216.251} C_DIS
LIN {X 0.152,Y -456.173,Z 1137.989,A 0.000,B 0.000,C 90.000,E1 213.992} C_DIS
LIN {X 0.123,Y -454.726,Z 1137.977,A 0.000,B 0.000,C 90.000,E1 211.750} C_DIS
LIN {X 0.079,Y -453.753,Z 1137.955,A 0.000,B 0.000,C 90.000,E1 207.897} C_DIS
LIN {X -0.098,Y -454.583,Z 1137.943,A 0.000,B 0.000,C 90.000,E1 205.668} C_DIS
LIN {X -0.234,Y -456.043,Z 1137.934,A 0.000,B 0.000,C 90.000,E1 204.079} C_DIS
LIN {X -0.201,Y -458.932,Z 1137.923,A 0.000,B 0.000,C 90.000,E1 202.153} C_DIS
LIN {X -0.264,Y -462.767,Z 1137.912,A 0.000,B 0.000,C 90.000,E1 200.248} C_DIS
LIN {X -0.015,Y -468.413,Z 1137.900,A 0.000,B 0.000,C 90.000,E1 198.000} C_DIS
LIN {X -0.169,Y -474.222,Z 1137.890,A 0.000,B 0.000,C 90.000,E1 196.134} C_DIS
LIN {X -0.169,Y -482.733,Z 1137.876,A 0.000,B 0.000,C 90.000,E1 193.647} C_DIS
LIN {X -0.012,Y -490.604,Z 1137.864,A 0.000,B 0.000,C 90.000,E1 191.478} C_DIS
LIN {X -0.136,Y -497.565,Z 1137.854,A 0.000,B 0.000,C 90.000,E1 189.670} C_DIS
LIN {X 0.056,Y -504.031,Z 1137.844,A 0.000,B 0.000,C 90.000,E1 187.992} C_DIS
LIN {X 0.057,Y -508.206,Z 1137.839,A 0.000,B 0.000,C 90.000,E1 186.947} C_DIS
LIN {X 0.109,Y -515.202,Z 1137.829,A 0.000,B 0.000,C 90.000,E1 185.163} C_DIS
LIN {X -0.237,Y -522.141,Z 1137.819,A 0.000,B 0.000,C 90.000,E1 183.440} C_DIS
LIN {X 0.171,Y -525.670,Z 1137.814,A 0.000,B 0.000,C 90.000,E1 182.522} C_DIS
LIN {X 0.011,Y -533.706,Z 1137.803,A 0.000,B 0.000,C 90.000,E1 180.516} C_DIS
LIN {X 0.027,Y -540.636,Z 1137.793,A 0.000,B 0.000,C 90.000,E1 178.797} C_DIS
LIN {X 0.137,Y -545.248,Z 1137.787,A 0.000,B 0.000,C 90.000,E1 177.650} C_DIS
LIN {X -0.135,Y -552.188,Z 1137.778,A 0.000,B 0.000,C 90.000,E1 175.988} C_DIS
LIN {X 0.247,Y -557.970,Z 1137.770,A 0.000,B 0.000,C 90.000,E1 174.552} C_DIS
LIN {X -0.169,Y -564.835,Z 1137.761,A 0.000,B 0.000,C 90.000,E1 172.932} C_DIS
LIN {X -0.051,Y -570.609,Z 1137.753,A 0.000,B 0.000,C 90.000,E1 171.546} C_DIS
LIN {X 0.256,Y -576.277,Z 1137.745,A 0.000,B 0.000,C 90.000,E1 170.151} C_DIS
LIN {X 0.220,Y -579.581,Z 1137.741,A 0.000,B 0.000,C 90.000,E1 169.342} C_DIS
LIN {X 0.222,Y -584.997,Z 1137.734,A 0.000,B 0.000,C 90.000,E1 167.993} C_DIS
LIN {X 0.066,Y -589.230,Z 1137.728,A 0.000,B 0.000,C 90.000,E1 166.937} C_DIS
LIN {X -0.038,Y -593.270,Z 1137.722,A 0.000,B 0.000,C 90.000,E1 165.880} C_DIS
LIN {X 0.059,Y -597.143,Z 1137.716,A 0.000,B 0.000,C 90.000,E1 164.810} C_DIS
LIN {X -0.073,Y -601.694,Z 1137.708,A 0.000,B 0.000,C 90.000,E1 163.504} C_DIS
LIN {X -0.230,Y -606.830,Z 1137.700,A 0.000,B 0.000,C 90.000,E1 161.945} C_DIS
LIN {X 0.168,Y -610.829,Z 1137.692,A 0.000,B 0.000,C 90.000,E1 160.604} C_DIS
LIN {X 0.115,Y -613.910,Z 1137.687,A 0.000,B 0.000,C 90.000,E1 159.571} C_DIS
LIN {X 0.065,Y -617.454,Z 1137.679,A 0.000,B 0.000,C 90.000,E1 158.284} C_DIS
LIN {X 0.055,Y -621.589,Z 1137.671,A 0.000,B 0.000,C 90.000,E1 156.741} C_DIS
LIN {X -0.192,Y -626.189,Z 1137.661,A 0.000,B 0.000,C 90.000,E1 154.973} C_DIS
LIN {X -0.104,Y -629.319,Z 1137.654,A 0.000,B 0.000,C 90.000,E1 153.691} C_DIS
LIN {X 0.041,Y -632.238,Z 1137.647,A 0.000,B 0.000,C 90.000,E1 152.410} C_DIS
LIN {X 0.224,Y -635.060,Z 1137.640,A 0.000,B 0.000,C 90.000,E1 151.129} C_DIS
LIN {X 0.198,Y -637.753,Z 1137.633,A 0.000,B 0.000,C 90.000,E1 149.871} C_DIS
LIN {X 0.216,Y -640.327,Z 1137.626,A 0.000,B 0.000,C 90.000,E1 148.614} C_DIS
LIN {X -0.330,Y -642.299,Z 1137.620,A 0.000,B 0.000,C 90.000,E1 147.661} C_DIS
LIN {X -0.030,Y -645.013,Z 1137.612,A 0.000,B 0.000,C 90.000,E1 146.135} C_DIS
LIN {X -0.042,Y -647.642,Z 1137.604,A 0.000,B 0.000,C 90.000,E1 144.642} C_DIS
LIN {X 0.213,Y -650.110,Z 1137.595,A 0.000,B 0.000,C 90.000,E1 143.130} C_DIS
LIN {X 0.014,Y -652.668,Z 1137.587,A 0.000,B 0.000,C 90.000,E1 141.662} C_DIS
LIN {X -0.229,Y -657.240,Z 1137.573,A 0.000,B 0.000,C 90.000,E1 139.218} C_DIS
LIN {X 0.101,Y -660.620,Z 1137.564,A 0.000,B 0.000,C 90.000,E1 137.472} C_DIS
LIN {X -0.006,Y -664.514,Z 1137.553,A 0.000,B 0.000,C 90.000,E1 135.526} C_DIS
LIN {X -0.007,Y -669.325,Z 1137.541,A 0.000,B 0.000,C 90.000,E1 133.338} C_DIS
LIN {X 0.120,Y -673.365,Z 1137.531,A 0.000,B 0.000,C 90.000,E1 131.634} C_DIS
LIN {X 0.307,Y -676.829,Z 1137.523,A 0.000,B 0.000,C 90.000,E1 130.172} C_DIS
LIN {X 0.302,Y -682.294,Z 1137.511,A 0.000,B 0.000,C 90.000,E1 128.016} C_DIS
LIN {X 0.322,Y -685.921,Z 1137.503,A 0.000,B 0.000,C 90.000,E1 126.583} C_DIS
LIN {X -0.215,Y -688.297,Z 1137.498,A 0.000,B 0.000,C 90.000,E1 125.678} C_DIS
LIN {X -0.091,Y -691.769,Z 1137.490,A 0.000,B 0.000,C 90.000,E1 124.246} C_DIS
LIN {X 0.243,Y -694.629,Z 1137.484,A 0.000,B 0.000,C 90.000,E1 123.038} C_DIS
LIN {X 0.050,Y -697.305,Z 1137.477,A 0.000,B 0.000,C 90.000,E1 121.878} C_DIS
LIN {X 0.229,Y -699.082,Z 1137.472,A 0.000,B 0.000,C 90.000,E1 120.924} C_DIS
LIN {X -0.271,Y -701.132,Z 1137.465,A 0.000,B 0.000,C 90.000,E1 119.795} C_DIS
LIN {X -0.131,Y -703.171,Z 1137.459,A 0.000,B 0.000,C 90.000,E1 118.615} C_DIS
LIN {X 0.091,Y -704.315,Z 1137.455,A 0.000,B 0.000,C 90.000,E1 117.897} C_DIS
LIN {X 0.001,Y -705.187,Z 1137.451,A 0.000,B 0.000,C 90.000,E1 117.206} C_DIS
LIN {X -0.048,Y -705.608,Z 1137.449,A 0.000,B 0.000,C 90.000,E1 116.744} C_DIS
LIN {X 0.175,Y -706.159,Z 1137.443,A 0.000,B 0.000,C 90.000,E1 115.796} C_DIS
LIN {X 0.116,Y -706.332,Z 1137.440,A 0.000,B 0.000,C 90.000,E1 115.103} C_DIS
LIN {X 0.062,Y -706.206,Z 1137.437,A 0.000,B 0.000,C 90.000,E1 114.643} C_DIS
LIN {X 0.353,Y -705.942,Z 1137.436,A 0.000,B 0.000,C 90.000,E1 114.387} C_DIS
LIN {X -0.001,Y -705.112,Z 1137.433,A 0.000,B 0.000,C 90.000,E1 113.951} C_DIS
LIN {X -0.358,Y -703.197,Z 1137.431,A 0.000,B 0.000,C 90.000,E1 113.515} C_DIS
LIN {X -0.076,Y -702.056,Z 1137.429,A 0.000,B 0.000,C 90.000,E1 113.259} C_DIS
LIN {X -0.095,Y -698.042,Z 1137.427,A 0.000,B 0.000,C 90.000,E1 112.823} C_DIS
LIN {X 0.036,Y -696.867,Z 1137.426,A 0.000,B 0.000,C 90.000,E1 112.695} C_DIS
LIN {X -0.101,Y -695.198,Z 1137.426,A 0.000,B 0.000,C 90.000,E1 112.589} C_DIS
LIN {X 0.254,Y -692.817,Z 1137.425,A 0.000,B 0.000,C 90.000,E1 112.461} C_DIS
LIN {X -0.174,Y -686.618,Z 1137.424,A 0.000,B 0.000,C 90.000,E1 112.280} C_DIS
LIN {X 0.126,Y -684.637,Z 1137.423,A 0.000,B 0.000,C 90.000,E1 112.206} C_DIS
LIN {X -0.176,Y -676.557,Z 1137.423,A 0.000,B 0.000,C 90.000,E1 112.153} C_DIS
LIN {X -0.205,Y -603.241,Z 1137.423,A 0.000,B 0.000,C 90.000,E1 112.153} C_DIS
LIN {X 0.195,Y -599.932,Z 1137.422,A 0.000,B 0.000,C 90.000,E1 111.897} C_DIS
LIN {X 0.239,Y -595.338,Z 1137.420,A 0.000,B 0.000,C 90.000,E1 111.535} C_DIS
LIN {X 0.019,Y -582.613,Z 1137.414,A 0.000,B 0.000,C 90.000,E1 110.429} C_DIS
LIN {X 0.158,Y -575.743,Z 1137.410,A 0.000,B 0.000,C 90.000,E1 109.812} C_DIS
LIN {X -0.179,Y -568.282,Z 1137.407,A 0.000,B 0.000,C 90.000,E1 109.268} C_DIS
LIN {X 0.030,Y -560.081,Z 1137.404,A 0.000,B 0.000,C 90.000,E1 108.725} C_DIS
LIN {X 0.200,Y -555.301,Z 1137.402,A 0.000,B 0.000,C 90.000,E1 108.417} C_DIS
LIN {X 0.315,Y -550.891,Z 1137.401,A 0.000,B 0.000,C 90.000,E1 108.055} C_DIS
LIN {X 0.243,Y -549.740,Z 1137.400,A 0.000,B 0.000,C 90.000,E1 107.873} C_DIS
LIN {X 0.202,Y -549.716,Z 1137.399,A 0.000,B 0.000,C 90.000,E1 107.873} C_DIS
LIN {X -0.067,Y -549.461,Z 1137.397,A 0.000,B 0.000,C 90.000,E1 107.511} C_DIS
LIN {X -0.190,Y -551.070,Z 1137.383,A 0.000,B 0.000,C 90.000,E1 105.009} C_DIS
LIN {X 0.087,Y -552.417,Z 1137.374,A 0.000,B 0.000,C 90.000,E1 103.300} C_DIS
LIN {X -0.266,Y -553.876,Z 1137.365,A 0.000,B 0.000,C 90.000,E1 101.658} C_DIS
LIN {X 0.080,Y -555.610,Z 1137.354,A 0.000,B 0.000,C 90.000,E1 99.670} C_DIS
LIN {X 0.093,Y -556.878,Z 1137.346,A 0.000,B 0.000,C 90.000,E1 98.276} C_DIS
LIN {X 0.048,Y -558.076,Z 1137.338,A 0.000,B 0.000,C 90.000,E1 96.891} C_DIS
LIN {X 0.097,Y -559.534,Z 1137.329,A 0.000,B 0.000,C 90.000,E1 95.220} C_DIS
LIN {X 0.043,Y -560.675,Z 1137.321,A 0.000,B 0.000,C 90.000,E1 93.841} C_DIS
LIN {X -0.027,Y -561.691,Z 1137.314,A 0.000,B 0.000,C 90.000,E1 92.465} C_DIS
LIN {X -0.178,Y -562.516,Z 1137.308,A 0.000,B 0.000,C 90.000,E1 91.375} C_DIS
LIN {X -0.123,Y -563.615,Z 1137.298,A 0.000,B 0.000,C 90.000,E1 89.714} C_DIS
LIN {X 0.195,Y -564.102,Z 1137.294,A 0.000,B 0.000,C 90.000,E1 88.854} C_DIS
LIN {X -0.272,Y -565.081,Z 1137.285,A 0.000,B 0.000,C 90.000,E1 87.249} C_DIS
LIN {X -0.122,Y -565.988,Z 1137.275,A 0.000,B 0.000,C 90.000,E1 85.584} C_DIS
LIN {X 0.099,Y -566.718,Z 1137.266,A 0.000,B 0.000,C 90.000,E1 83.913} C_DIS
LIN {X -0.058,Y -567.631,Z 1137.256,A 0.000,B 0.000,C 90.000,E1 82.008} C_DIS
LIN {X 0.085,Y -568.262,Z 1137.248,A 0.000,B 0.000,C 90.000,E1 80.622} C_DIS
LIN {X -0.058,Y -568.960,Z 1137.239,A 0.000,B 0.000,C 90.000,E1 78.993} C_DIS
LIN {X -0.077,Y -569.768,Z 1137.230,A 0.000,B 0.000,C 90.000,E1 77.353} C_DIS
LIN {X 0.053,Y -570.528,Z 1137.221,A 0.000,B 0.000,C 90.000,E1 75.700} C_DIS
LIN {X -0.014,Y -571.582,Z 1137.210,A 0.000,B 0.000,C 90.000,E1 73.795} C_DIS
LIN {X 0.127,Y -572.464,Z 1137.202,A 0.000,B 0.000,C 90.000,E1 72.417} C_DIS
LIN {X 0.095,Y -573.680,Z 1137.193,A 0.000,B 0.000,C 90.000,E1 70.786} C_DIS
LIN {X 0.279,Y -575.503,Z 1137.181,A 0.000,B 0.000,C 90.000,E1 68.592} C_DIS
LIN {X 0.178,Y -577.067,Z 1137.172,A 0.000,B 0.000,C 90.000,E1 66.975} C_DIS
LIN {X -0.273,Y -578.247,Z 1137.165,A 0.000,B 0.000,C 90.000,E1 65.665} C_DIS
LIN {X 0.057,Y -579.507,Z 1137.157,A 0.000,B 0.000,C 90.000,E1 64.280} C_DIS
LIN {X 0.006,Y -580.895,Z 1137.148,A 0.000,B 0.000,C 90.000,E1 62.666} C_DIS
LIN {X -0.014,Y -582.226,Z 1137.139,A 0.000,B 0.000,C 90.000,E1 61.051} C_DIS
LIN {X -0.103,Y -583.187,Z 1137.132,A 0.000,B 0.000,C 90.000,E1 59.715} C_DIS
LIN {X 0.328,Y -584.113,Z 1137.124,A 0.000,B 0.000,C 90.000,E1 58.329} C_DIS
LIN {X -0.046,Y -585.069,Z 1137.115,A 0.000,B 0.000,C 90.000,E1 56.755} C_DIS
LIN {X 0.077,Y -586.010,Z 1137.106,A 0.000,B 0.000,C 90.000,E1 55.135} C_DIS
LIN {X -0.074,Y -586.907,Z 1137.097,A 0.000,B 0.000,C 90.000,E1 53.543} C_DIS
LIN {X 0.156,Y -587.283,Z 1137.093,A 0.000,B 0.000,C 90.000,E1 52.718} C_DIS
LIN {X 0.208,Y -587.887,Z 1137.086,A 0.000,B 0.000,C 90.000,E1 51.376} C_DIS
LIN {X -0.032,Y -588.239,Z 1137.081,A 0.000,B 0.000,C 90.000,E1 50.598} C_DIS
LIN {X 0.099,Y -588.492,Z 1137.077,A 0.000,B 0.000,C 90.000,E1 49.784} C_DIS
LIN {X 0.114,Y -588.627,Z 1137.069,A 0.000,B 0.000,C 90.000,E1 48.447} C_DIS
LIN {X -0.066,Y -588.521,Z 1137.060,A 0.000,B 0.000,C 90.000,E1 46.863} C_DIS
LIN {X -0.221,Y -588.299,Z 1137.054,A 0.000,B 0.000,C 90.000,E1 45.810} C_DIS
LIN {X 0.041,Y -587.940,Z 1137.048,A 0.000,B 0.000,C 90.000,E1 44.717} C_DIS
LIN {X 0.299,Y -587.372,Z 1137.043,A 0.000,B 0.000,C 90.000,E1 43.623} C_DIS
LIN {X -0.023,Y -586.890,Z 1137.038,A 0.000,B 0.000,C 90.000,E1 42.852} C_DIS
LIN {X -0.093,Y -586.362,Z 1137.035,A 0.000,B 0.000,C 90.000,E1 42.324} C_DIS
LIN {X 0.046,Y -586.229,Z 1137.034,A 0.000,B 0.000,C 90.000,E1 42.043} C_DIS
LIN {X 0.071,Y -584.719,Z 1137.026,A 0.000,B 0.000,C 90.000,E1 40.701} C_DIS
LIN {X -0.099,Y -583.392,Z 1137.020,A 0.000,B 0.000,C 90.000,E1 39.644} C_DIS
LIN {X -0.120,Y -581.458,Z 1137.013,A 0.000,B 0.000,C 90.000,E1 38.302} C_DIS
LIN {X -0.246,Y -579.567,Z 1137.007,A 0.000,B 0.000,C 90.000,E1 37.237} C_DIS
LIN {X 0.253,Y -577.915,Z 1137.002,A 0.000,B 0.000,C 90.000,E1 36.377} C_DIS
LIN {X -0.073,Y -575.952,Z 1136.998,A 0.000,B 0.000,C 90.000,E1 35.598} C_DIS
LIN {X 0.232,Y -574.502,Z 1136.995,A 0.000,B 0.000,C 90.000,E1 35.025} C_DIS
LIN {X -0.134,Y -572.052,Z 1136.990,A 0.000,B 0.000,C 90.000,E1 34.246} C_DIS
LIN {X -0.183,Y -570.255,Z 1136.987,A 0.000,B 0.000,C 90.000,E1 33.706} C_DIS
LIN {X -0.119,Y -567.124,Z 1136.983,A 0.000,B 0.000,C 90.000,E1 32.880} C_DIS
LIN {X -0.093,Y -563.790,Z 1136.978,A 0.000,B 0.000,C 90.000,E1 32.054} C_DIS
LIN {X -0.026,Y -559.305,Z 1136.973,A 0.000,B 0.000,C 90.000,E1 31.082} C_DIS
LIN {X -0.095,Y -555.002,Z 1136.968,A 0.000,B 0.000,C 90.000,E1 30.256} C_DIS
LIN {X 0.103,Y -551.170,Z 1136.964,A 0.000,B 0.000,C 90.000,E1 29.539} C_DIS
LIN {X -0.095,Y -547.975,Z 1136.961,A 0.000,B 0.000,C 90.000,E1 28.999} C_DIS
LIN {X -0.218,Y -541.742,Z 1136.956,A 0.000,B 0.000,C 90.000,E1 28.025} C_DIS
LIN {X -0.142,Y -536.855,Z 1136.952,A 0.000,B 0.000,C 90.000,E1 27.308} C_DIS
LIN {X -0.214,Y -532.643,Z 1136.948,A 0.000,B 0.000,C 90.000,E1 26.744} C_DIS
LIN {X -0.055,Y -524.715,Z 1136.943,A 0.000,B 0.000,C 90.000,E1 25.720} C_DIS
LIN {X -0.099,Y -515.950,Z 1136.937,A 0.000,B 0.000,C 90.000,E1 24.719} C_DIS
LIN {X -0.178,Y -509.583,Z 1136.933,A 0.000,B 0.000,C 90.000,E1 24.027} C_DIS
LIN {X -0.205,Y -504.104,Z 1136.930,A 0.000,B 0.000,C 90.000,E1 23.462} C_DIS
LIN {X 0.134,Y -495.772,Z 1136.926,A 0.000,B 0.000,C 90.000,E1 22.589} C_DIS
LIN {X 0.204,Y -487.113,Z 1136.921,A 0.000,B 0.000,C 90.000,E1 21.770} C_DIS
LIN {X 0.154,Y -478.350,Z 1136.917,A 0.000,B 0.000,C 90.000,E1 20.972} C_DIS
LIN {X 0.078,Y -466.576,Z 1136.911,A 0.000,B 0.000,C 90.000,E1 19.939} C_DIS
LIN {X 0.241,Y -451.840,Z 1136.904,A 0.000,B 0.000,C 90.000,E1 18.598} C_DIS
LIN {X -0.004,Y -434.562,Z 1136.894,A 0.000,B 0.000,C 90.000,E1 16.985} C_DIS
LIN {X -0.157,Y -421.791,Z 1136.887,A 0.000,B 0.000,C 90.000,E1 15.662} C_DIS
LIN {X 0.008,Y -410.713,Z 1136.880,A 0.000,B 0.000,C 90.000,E1 14.356} C_DIS
LIN {X -0.146,Y -402.838,Z 1136.874,A 0.000,B 0.000,C 90.000,E1 13.355} C_DIS
LIN {X -0.069,Y -398.158,Z 1136.870,A 0.000,B 0.000,C 90.000,E1 12.647} C_DIS
LIN {X 0.131,Y -394.779,Z 1136.867,A 0.000,B 0.000,C 90.000,E1 12.007} C_DIS
LIN {X 0.120,Y -392.908,Z 1136.864,A 0.000,B 0.000,C 90.000,E1 11.478} C_DIS
LIN {X 0.094,Y -392.158,Z 1136.861,A 0.000,B 0.000,C 90.000,E1 10.950} C_DIS
LIN {X 0.007,Y -392.800,Z 1136.857,A 0.000,B 0.000,C 90.000,E1 10.254} C_DIS
LIN {X -0.002,Y -394.159,Z 1136.853,A 0.000,B 0.000,C 90.000,E1 9.557} C_DIS
LIN {X -0.144,Y -398.074,Z 1136.845,A 0.000,B 0.000,C 90.000,E1 8.163} C_DIS
LIN {X 0.092,Y -403.052,Z 1136.837,A 0.000,B 0.000,C 90.000,E1 6.549} C_DIS
LIN {X 0.061,Y -405.086,Z 1136.834,A 0.000,B 0.000,C 90.000,E1 6.030} C_DIS
LIN {X 0.013,Y -407.138,Z 1136.831,A 0.000,B 0.000,C 90.000,E1 5.625} C_DIS
LIN {X -0.005,Y -408.253,Z 1136.830,A 0.000,B 0.000,C 90.000,E1 5.454} C_DIS
LIN {X 0.058,Y -411.383,Z 1136.828,A 0.000,B 0.000,C 90.000,E1 5.049} C_DIS
LIN {X 0.001,Y -417.705,Z 1136.825,A 0.000,B 0.000,C 90.000,E1 4.531} C_DIS
LIN {X -0.067,Y -425.133,Z 1136.822,A 0.000,B 0.000,C 90.000,E1 4.012} C_DIS
LIN {X -0.017,Y -449.604,Z 1136.813,A 0.000,B 0.000,C 90.000,E1 2.293} C_DIS
LIN {X 0.079,Y -464.059,Z 1136.807,A 0.000,B 0.000,C 90.000,E1 1.318} C_DIS
LIN {X -0.047,Y -472.159,Z 1136.804,A 0.000,B 0.000,C 90.000,E1 0.802} C_DIS
LIN {X -0.238,Y -481.797,Z 1136.801,A 0.000,B 0.000,C 90.000,E1 0.172} C_DIS
LIN {X 0.238,Y -491.430,Z 1136.797,A 0.000,B 0.000,C 90.000,E1 359.427} C_DIS
LIN {X 0.233,Y -497.449,Z 1136.794,A 0.000,B 0.000,C 90.000,E1 358.969} C_DIS
LIN {X 0.072,Y -503.409,Z 1136.792,A 0.000,B 0.000,C 90.000,E1 358.511} C_DIS
LIN {X 0.132,Y -510.542,Z 1136.788,A 0.000,B 0.000,C 90.000,E1 357.879} C_DIS
LIN {X -0.099,Y -517.469,Z 1136.785,A 0.000,B 0.000,C 90.000,E1 357.249} C_DIS
LIN {X -0.004,Y -521.330,Z 1136.782,A 0.000,B 0.000,C 90.000,E1 356.846} C_DIS
LIN {X -0.225,Y -527.727,Z 1136.779,A 0.000,B 0.000,C 90.000,E1 356.159} C_DIS
LIN {X 0.245,Y -533.461,Z 1136.775,A 0.000,B 0.000,C 90.000,E1 355.412} C_DIS
LIN {X 0.264,Y -537.796,Z 1136.771,A 0.000,B 0.000,C 90.000,E1 354.837} C_DIS
LIN {X 0.050,Y -542.546,Z 1136.768,A 0.000,B 0.000,C 90.000,E1 354.147} C_DIS
LIN {X 0.134,Y -546.101,Z 1136.764,A 0.000,B 0.000,C 90.000,E1 353.571} C_DIS
LIN {X 0.051,Y -550.079,Z 1136.760,A 0.000,B 0.000,C 90.000,E1 352.875} C_DIS
LIN {X -0.243,Y -554.383,Z 1136.756,A 0.000,B 0.000,C 90.000,E1 352.064} C_DIS
LIN {X 0.178,Y -556.398,Z 1136.754,A 0.000,B 0.000,C 90.000,E1 351.602} C_DIS
LIN {X 0.196,Y -559.344,Z 1136.750,A 0.000,B 0.000,C 90.000,E1 350.905} C_DIS
LIN {X -0.012,Y -562.547,Z 1136.745,A 0.000,B 0.000,C 90.000,E1 350.095} C_DIS
LIN {X -0.195,Y -565.510,Z 1136.740,A 0.000,B 0.000,C 90.000,E1 349.285} C_DIS
LIN {X -0.069,Y -569.104,Z 1136.734,A 0.000,B 0.000,C 90.000,E1 348.173} C_DIS
LIN {X -0.259,Y -573.168,Z 1136.727,A 0.000,B 0.000,C 90.000,E1 346.825} C_DIS
LIN {X -0.244,Y -576.880,Z 1136.719,A 0.000,B 0.000,C 90.000,E1 345.463} C_DIS
LIN {X 0.183,Y -579.704,Z 1136.713,A 0.000,B 0.000,C 90.000,E1 344.338} C_DIS
LIN {X -0.082,Y -583.101,Z 1136.706,A 0.000,B 0.000,C 90.000,E1 343.015} C_DIS
LIN {X 0.273,Y -586.354,Z 1136.698,A 0.000,B 0.000,C 90.000,E1 341.638} C_DIS
LIN {X 0.116,Y -589.213,Z 1136.691,A 0.000,B 0.000,C 90.000,E1 340.315} C_DIS
LIN {X 0.090,Y -590.787,Z 1136.686,A 0.000,B 0.000,C 90.000,E1 339.518} C_DIS
LIN {X -0.029,Y -592.755,Z 1136.680,A 0.000,B 0.000,C 90.000,E1 338.465} C_DIS
LIN {X -0.016,Y -593.959,Z 1136.676,A 0.000,B 0.000,C 90.000,E1 337.667} C_DIS
LIN {X -0.183,Y -595.525,Z 1136.669,A 0.000,B 0.000,C 90.000,E1 336.357} C_DIS
LIN {X 0.092,Y -596.200,Z 1136.664,A 0.000,B 0.000,C 90.000,E1 335.537} C_DIS
LIN {X 0.293,Y -596.830,Z 1136.658,A 0.000,B 0.000,C 90.000,E1 334.460} C_DIS
LIN {X 0.047,Y -596.950,Z 1136.654,A 0.000,B 0.000,C 90.000,E1 333.691} C_DIS
LIN {X -0.116,Y -596.847,Z 1136.651,A 0.000,B 0.000,C 90.000,E1 333.179} C_DIS
LIN {X 0.081,Y -596.151,Z 1136.645,A 0.000,B 0.000,C 90.000,E1 332.103} C_DIS
LIN {X 0.192,Y -595.650,Z 1136.642,A 0.000,B 0.000,C 90.000,E1 331.563} C_DIS
LIN {X -0.168,Y -594.163,Z 1136.636,A 0.000,B 0.000,C 90.000,E1 330.539} C_DIS
LIN {X 0.036,Y -591.884,Z 1136.630,A 0.000,B 0.000,C 90.000,E1 329.459} C_DIS
LIN {X -0.175,Y -590.468,Z 1136.627,A 0.000,B 0.000,C 90.000,E1 328.948} C_DIS
LIN {X -0.093,Y -588.713,Z 1136.625,A 0.000,B 0.000,C 90.000,E1 328.408} C_DIS
LIN {X -0.022,Y -586.814,Z 1136.622,A 0.000,B 0.000,C 90.000,E1 327.867} C_DIS
LIN {X -0.032,Y -584.037,Z 1136.618,A 0.000,B 0.000,C 90.000,E1 327.199} C_DIS
LIN {X 0.168,Y -579.974,Z 1136.613,A 0.000,B 0.000,C 90.000,E1 326.373} C_DIS
LIN {X -0.067,Y -576.102,Z 1136.610,A 0.000,B 0.000,C 90.000,E1 325.722} C_DIS
LIN {X -0.001,Y -573.732,Z 1136.607,A 0.000,B 0.000,C 90.000,E1 325.308} C_DIS
LIN {X 0.188,Y -569.221,Z 1136.604,A 0.000,B 0.000,C 90.000,E1 324.609} C_DIS
LIN {X 0.334,Y -564.301,Z 1136.600,A 0.000,B 0.000,C 90.000,E1 323.909} C_DIS
LIN {X -0.119,Y -561.141,Z 1136.597,A 0.000,B 0.000,C 90.000,E1 323.543} C_DIS
LIN {X 0.077,Y -556.481,Z 1136.594,A 0.000,B 0.000,C 90.000,E1 322.970} C_DIS
LIN {X -0.035,Y -549.181,Z 1136.590,A 0.000,B 0.000,C 90.000,E1 322.145} C_DIS
LIN {X -0.073,Y -540.340,Z 1136.584,A 0.000,B 0.000,C 90.000,E1 321.170} C_DIS
LIN {X 0.079,Y -535.405,Z 1136.581,A 0.000,B 0.000,C 90.000,E1 320.598} C_DIS
LIN {X -0.097,Y -532.121,Z 1136.579,A 0.000,B 0.000,C 90.000,E1 320.194} C_DIS
LIN {X 0.053,Y -529.789,Z 1136.577,A 0.000,B 0.000,C 90.000,E1 319.828} C_DIS
LIN {X -0.125,Y -528.971,Z 1136.576,A 0.000,B 0.000,C 90.000,E1 319.703} C_DIS
LIN {X -0.032,Y -527.356,Z 1136.574,A 0.000,B 0.000,C 90.000,E1 319.337} C_DIS
LIN {X 0.173,Y -525.307,Z 1136.571,A 0.000,B 0.000,C 90.000,E1 318.690} C_DIS
LIN {X -0.019,Y -524.959,Z 1136.570,A 0.000,B 0.000,C 90.000,E1 318.566} C_DIS
LIN {X -0.301,Y -524.236,Z 1136.567,A 0.000,B 0.000,C 90.000,E1 318.162} C_DIS
LIN {X 0.004,Y -523.747,Z 1136.566,A 0.000,B 0.000,C 90.000,E1 317.838} C_DIS
LIN {X -0.078,Y -523.160,Z 1136.562,A 0.000,B 0.000,C 90.000,E1 317.067} C_DIS
LIN {X 0.064,Y -523.493,Z 1136.547,A 0.000,B 0.000,C 90.000,E1 314.433} C_DIS
LIN {X 0.098,Y -523.815,Z 1136.539,A 0.000,B 0.000,C 90.000,E1 312.975} C_DIS
LIN {X -0.071,Y -524.771,Z 1136.524,A 0.000,B 0.000,C 90.000,E1 310.378} C_DIS
LIN {X 0.073,Y -525.546,Z 1136.516,A 0.000,B 0.000,C 90.000,E1 308.910} C_DIS
LIN {X 0.176,Y -526.801,Z 1136.505,A 0.000,B 0.000,C 90.000,E1 306.870} C_DIS
LIN {X 0.007,Y -527.948,Z 1136.495,A 0.000,B 0.000,C 90.000,E1 305.152} C_DIS
LIN {X -0.015,Y -529.109,Z 1136.486,A 0.000,B 0.000,C 90.000,E1 303.420} C_DIS
LIN {X 0.034,Y -529.844,Z 1136.479,A 0.000,B 0.000,C 90.000,E1 302.260} C_DIS
LIN {X -0.060,Y -531.223,Z 1136.470,A 0.000,B 0.000,C 90.000,E1 300.541} C_DIS
LIN {X -0.114,Y -532.412,Z 1136.460,A 0.000,B 0.000,C 90.000,E1 298.821} C_DIS
LIN {X 0.168,Y -533.041,Z 1136.454,A 0.000,B 0.000,C 90.000,E1 297.641} C_DIS
LIN {X 0.213,Y -533.524,Z 1136.447,A 0.000,B 0.000,C 90.000,E1 296.488} C_DIS
LIN {X -0.024,Y -533.830,Z 1136.439,A 0.000,B 0.000,C 90.000,E1 295.079} C_DIS
LIN {X 0.002,Y -533.893,Z 1136.431,A 0.000,B 0.000,C 90.000,E1 293.643} C_DIS
LIN {X 0.030,Y -533.870,Z 1136.423,A 0.000,B 0.000,C 90.000,E1 292.206} C_DIS
LIN {X 0.149,Y -533.828,Z 1136.417,A 0.000,B 0.000,C 90.000,E1 291.046} C_DIS
LIN {X -0.028,Y -533.659,Z 1136.409,A 0.000,B 0.000,C 90.000,E1 289.631} C_DIS
LIN {X 0.112,Y -533.376,Z 1136.401,A 0.000,B 0.000,C 90.000,E1 288.181} C_DIS
LIN {X -0.232,Y -532.824,Z 1136.392,A 0.000,B 0.000,C 90.000,E1 286.496} C_DIS
LIN {X 0.026,Y -532.489,Z 1136.387,A 0.000,B 0.000,C 90.000,E1 285.607} C_DIS
LIN {X -0.022,Y -531.735,Z 1136.379,A 0.000,B 0.000,C 90.000,E1 284.175} C_DIS
LIN {X 0.178,Y -531.006,Z 1136.371,A 0.000,B 0.000,C 90.000,E1 282.715} C_DIS
LIN {X -0.036,Y -530.279,Z 1136.363,A 0.000,B 0.000,C 90.000,E1 281.299} C_DIS
LIN {X 0.111,Y -529.108,Z 1136.352,A 0.000,B 0.000,C 90.000,E1 279.265} C_DIS
LIN {X 0.128,Y -528.112,Z 1136.342,A 0.000,B 0.000,C 90.000,E1 277.530} C_DIS
LIN {X 0.122,Y -527.260,Z 1136.332,A 0.000,B 0.000,C 90.000,E1 275.796} C_DIS
LIN {X 0.030,Y -526.635,Z 1136.324,A 0.000,B 0.000,C 90.000,E1 274.359} C_DIS
LIN {X -0.078,Y -526.002,Z 1136.316,A 0.000,B 0.000,C 90.000,E1 272.922} C_DIS
LIN {X 0.262,Y -525.287,Z 1136.307,A 0.000,B 0.000,C 90.000,E1 271.146} C_DIS
LIN {X 0.054,Y -524.534,Z 1136.297,A 0.000,B 0.000,C 90.000,E1 269.427} C_DIS
LIN {X -0.158,Y -523.712,Z 1136.287,A 0.000,B 0.000,C 90.000,E1 267.707} C_DIS
LIN {X 0.221,Y -523.068,Z 1136.281,A 0.000,B 0.000,C 90.000,E1 266.502} C_DIS
LIN {X 0.055,Y -522.288,Z 1136.273,A 0.000,B 0.000,C 90.000,E1 265.065} C_DIS
LIN {X -0.063,Y -521.738,Z 1136.268,A 0.000,B 0.000,C 90.000,E1 264.204} C_DIS
LIN {X -0.201,Y -520.685,Z 1136.261,A 0.000,B 0.000,C 90.000,E1 263.053} C_DIS
LIN {X 0.218,Y -519.255,Z 1136.253,A 0.000,B 0.000,C 90.000,E1 261.546} C_DIS
LIN {X 0.085,Y -517.188,Z 1136.242,A 0.000,B 0.000,C 90.000,E1 259.511} C_DIS
LIN {X 0.012,Y -515.371,Z 1136.232,A 0.000,B 0.000,C 90.000,E1 257.757} C_DIS
LIN {X -0.066,Y -514.267,Z 1136.225,A 0.000,B 0.000,C 90.000,E1 256.589} C_DIS
LIN {X -0.011,Y -512.466,Z 1136.214,A 0.000,B 0.000,C 90.000,E1 254.519} C_DIS
LIN {X 0.074,Y -511.054,Z 1136.206,A 0.000,B 0.000,C 90.000,E1 253.032} C_DIS
LIN {X 0.000,Y -508.973,Z 1136.194,A 0.000,B 0.000,C 90.000,E1 250.967} C_DIS
LIN {X -0.314,Y -507.307,Z 1136.186,A 0.000,B 0.000,C 90.000,E1 249.518} C_DIS
LIN {X 0.073,Y -506.051,Z 1136.179,A 0.000,B 0.000,C 90.000,E1 248.284} C_DIS
LIN {X 0.064,Y -504.351,Z 1136.171,A 0.000,B 0.000,C 90.000,E1 246.794} C_DIS
LIN {X 0.016,Y -502.468,Z 1136.163,A 0.000,B 0.000,C 90.000,E1 245.305} C_DIS
LIN {X -0.035,Y -499.984,Z 1136.153,A 0.000,B 0.000,C 90.000,E1 243.512} C_DIS
LIN {X -0.186,Y -497.784,Z 1136.145,A 0.000,B 0.000,C 90.000,E1 242.025} C_DIS
LIN {X -0.109,Y -494.941,Z 1136.134,A 0.000,B 0.000,C 90.000,E1 240.205} C_DIS
LIN {X 0.130,Y -492.413,Z 1136.126,A 0.000,B 0.000,C 90.000,E1 238.663} C_DIS
LIN {X -0.092,Y -490.004,Z 1136.118,A 0.000,B 0.000,C 90.000,E1 237.168} C_DIS
LIN {X 0.148,Y -486.975,Z 1136.107,A 0.000,B 0.000,C 90.000,E1 235.308} C_DIS
LIN {X -0.088,Y -483.936,Z 1136.097,A 0.000,B 0.000,C 90.000,E1 233.497} C_DIS
LIN {X -0.013,Y -480.227,Z 1136.085,A 0.000,B 0.000,C 90.000,E1 231.331} C_DIS
LIN {X 0.089,Y -476.844,Z 1136.075,A 0.000,B 0.000,C 90.000,E1 229.461} C_DIS
LIN {X -0.243,Y -473.612,Z 1136.065,A 0.000,B 0.000,C 90.000,E1 227.634} C_DIS
LIN {X 0.161,Y -469.257,Z 1136.051,A 0.000,B 0.000,C 90.000,E1 225.081} C_DIS
LIN {X 0.028,Y -465.947,Z 1136.038,A 0.000,B 0.000,C 90.000,E1 222.894} C_DIS
LIN {X -0.001,Y -464.228,Z 1136.031,A 0.000,B 0.000,C 90.000,E1 221.634} C_DIS
LIN {X -0.162,Y -461.075,Z 1136.017,A 0.000,B 0.000,C 90.000,E1 219.116} C_DIS
LIN {X 0.084,Y -458.018,Z 1136.001,A 0.000,B 0.000,C 90.000,E1 216.217} C_DIS
LIN {X -0.140,Y -456.136,Z 1135.991,A 0.000,B 0.000,C 90.000,E1 214.326} C_DIS
LIN {X -0.278,Y -454.683,Z 1135.980,A 0.000,B 0.000,C 90.000,E1 212.418} C_DIS
LIN {X 0.099,Y -453.153,Z 1135.962,A 0.000,B 0.000,C 90.000,E1 209.155} C_DIS
LIN {X -0.173,Y -453.069,Z 1135.951,A 0.000,B 0.000,C 90.000,E1 207.257} C_DIS
LIN {X 0.264,Y -453.679,Z 1135.942,A 0.000,B 0.000,C 90.000,E1 205.591} C_DIS
LIN {X -0.079,Y -455.069,Z 1135.933,A 0.000,B 0.000,C 90.000,E1 204.027} C_DIS
LIN {X 0.125,Y -456.901,Z 1135.926,A 0.000,B 0.000,C 90.000,E1 202.717} C_DIS
LIN {X -0.160,Y -459.767,Z 1135.917,A 0.000,B 0.000,C 90.000,E1 201.153} C_DIS
LIN {X -0.003,Y -464.936,Z 1135.905,A 0.000,B 0.000,C 90.000,E1 198.906} C_DIS
LIN {X 0.161,Y -471.338,Z 1135.893,A 0.000,B 0.000,C 90.000,E1 196.677} C_DIS
LIN {X -0.058,Y -477.654,Z 1135.882,A 0.000,B 0.000,C 90.000,E1 194.828} C_DIS
LIN {X -0.190,Y -487.682,Z 1135.867,A 0.000,B 0.000,C 90.000,E1 192.063} C_DIS
LIN {X 0.007,Y -495.844,Z 1135.855,A 0.000,B 0.000,C 90.000,E1 189.905} C_DIS
LIN {X -0.005,Y -501.769,Z 1135.847,A 0.000,B 0.000,C 90.000,E1 188.398} C_DIS
LIN {X 0.094,Y -507.751,Z 1135.838,A 0.000,B 0.000,C 90.000,E1 186.891} C_DIS
LIN {X -0.072,Y -514.178,Z 1135.829,A 0.000,B 0.000,C 90.000,E1 185.277} C_DIS
LIN {X -0.089,Y -519.423,Z 1135.822,A 0.000,B 0.000,C 90.000,E1 183.955} C_DIS
LIN {X 0.192,Y -525.359,Z 1135.814,A 0.000,B 0.000,C 90.000,E1 182.465} C_DIS
LIN {X 0.038,Y -532.294,Z 1135.804,A 0.000,B 0.000,C 90.000,E1 180.745} C_DIS
LIN {X 0.035,Y -540.419,Z 1135.793,A 0.000,B 0.000,C 90.000,E1 178.740} C_DIS
LIN {X 0.141,Y -545.066,Z 1135.787,A 0.000,B 0.000,C 90.000,E1 177.593} C_DIS
LIN {X -0.096,Y -552.074,Z 1135.777,A 0.000,B 0.000,C 90.000,E1 175.927} C_DIS
LIN {X 0.296,Y -557.920,Z 1135.770,A 0.000,B 0.000,C 90.000,E1 174.489} C_DIS
LIN {X -0.090,Y -566.023,Z 1135.759,A 0.000,B 0.000,C 90.000,E1 172.591} C_DIS
LIN {X 0.126,Y -571.801,Z 1135.751,A 0.000,B 0.000,C 90.000,E1 171.197} C_DIS
LIN {X -0.112,Y -577.527,Z 1135.744,A 0.000,B 0.000,C 90.000,E1 169.859} C_DIS
LIN {X -0.024,Y -584.054,Z 1135.735,A 0.000,B 0.000,C 90.000,E1 168.229} C_DIS
LIN {X 0.057,Y -589.380,Z 1135.727,A 0.000,B 0.000,C 90.000,E1 166.881} C_DIS
LIN {X -0.313,Y -592.429,Z 1135.723,A 0.000,B 0.000,C 90.000,E1 166.117} C_DIS
LIN {X -0.230,Y -596.365,Z 1135.717,A 0.000,B 0.000,C 90.000,E1 165.046} C_DIS
LIN {X 0.202,Y -600.983,Z 1135.709,A 0.000,B 0.000,C 90.000,E1 163.685} C_DIS
LIN {X 0.031,Y -606.150,Z 1135.701,A 0.000,B 0.000,C 90.000,E1 162.127} C_DIS
LIN {X -0.358,Y -610.225,Z 1135.693,A 0.000,B 0.000,C 90.000,E1 160.859} C_DIS
LIN {X 0.099,Y -614.062,Z 1135.686,A 0.000,B 0.000,C 90.000,E1 159.518} C_DIS
LIN {X 0.048,Y -617.602,Z 1135.679,A 0.000,B 0.000,C 90.000,E1 158.230} C_DIS
LIN {X 0.279,Y -621.707,Z 1135.671,A 0.000,B 0.000,C 90.000,E1 156.666} C_DIS
LIN {X 0.036,Y -625.659,Z 1135.662,A 0.000,B 0.000,C 90.000,E1 155.153} C_DIS
LIN {X -0.156,Y -628.807,Z 1135.655,A 0.000,B 0.000,C 90.000,E1 153.896} C_DIS
LIN {X -0.056,Y -631.132,Z 1135.649,A 0.000,B 0.000,C 90.000,E1 152.871} C_DIS
LIN {X 0.107,Y -634.004,Z 1135.642,A 0.000,B 0.000,C 90.000,E1 151.591} C_DIS
LIN {X 0.061,Y -636.744,Z 1135.635,A 0.000,B 0.000,C 90.000,E1 150.333} C_DIS
LIN {X 0.112,Y -639.876,Z 1135.627,A 0.000,B 0.000,C 90.000,E1 148.820} C_DIS
LIN {X -0.046,Y -642.336,Z 1135.620,A 0.000,B 0.000,C 90.000,E1 147.582} C_DIS
LIN {X -0.153,Y -644.607,Z 1135.613,A 0.000,B 0.000,C 90.000,E1 146.342} C_DIS
LIN {X -0.273,Y -647.674,Z 1135.603,A 0.000,B 0.000,C 90.000,E1 144.609} C_DIS
LIN {X 0.077,Y -649.727,Z 1135.596,A 0.000,B 0.000,C 90.000,E1 143.336} C_DIS
LIN {X -0.083,Y -652.710,Z 1135.587,A 0.000,B 0.000,C 90.000,E1 141.618} C_DIS
LIN {X 0.087,Y -657.281,Z 1135.573,A 0.000,B 0.000,C 90.000,E1 139.138} C_DIS
LIN {X 0.421,Y -660.647,Z 1135.563,A 0.000,B 0.000,C 90.000,E1 137.391} C_DIS
LIN {X -0.148,Y -664.048,Z 1135.554,A 0.000,B 0.000,C 90.000,E1 135.729} C_DIS
LIN {X -0.172,Y -668.838,Z 1135.542,A 0.000,B 0.000,C 90.000,E1 133.542} C_DIS
